LIN {X 0,Y 224.89,Z 892.917,A -85,B 0,C 180,E1 -24408.732,E2 -24408.732} C_VEL
LIN {X 0,Y 229.595,Z 886.207,A -85,B 0,C 180,E1 -24414.165,E2 -24414.165} C_VEL
LIN {X 0,Y 235.615,Z 877.788,A -85,B 0,C 180,E1 -24419.211,E2 -24419.211} C_VEL
LIN {X 0,Y 242.277,Z 868.356,A -85,B 0,C 180,E1 -24423.575,E2 -24423.575} C_VEL
LIN {X 0,Y 250.04,Z 856.97,A -85,B 0,C 180,E1 -24427.722,E2 -24427.722} C_VEL
LIN {X 0,Y 258.343,Z 844.109,A -85,B 0,C 180,E1 -24431.44,E2 -24431.44} C_VEL
LIN {X 0,Y 266.959,Z 829.748,A -85,B 0,C 180,E1 -24434.761,E2 -24434.761} C_VEL
LIN {X 0,Y 275.684,Z 813.801,A -85,B 0,C 180,E1 -24437.722,E2 -24437.722} C_VEL
LIN {X 0,Y 283.965,Z 796.943,A -85,B 0,C 180,E1 -24440.246,E2 -24440.246} C_VEL
LIN {X 0,Y 291.586,Z 779.329,A -85,B 0,C 180,E1 -24442.385,E2 -24442.385} C_VEL
LIN {X 0,Y 298.391,Z 761.127,A -85,B 0,C 180,E1 -24444.186,E2 -24444.186} C_VEL
LIN {X 0,Y 304.38,Z 742.174,A -85,B 0,C 180,E1 -24445.708,E2 -24445.708} C_VEL
LIN {X 0,Y 309.449,Z 722.453,A -85,B 0,C 180,E1 -24446.981,E2 -24446.981} C_VEL
LIN {X 0,Y 313.937,Z 699.919,A -85,B 0,C 180,E1 -24448.124,E2 -24448.124} C_VEL
LIN {X 0,Y 321.08,Z 660.976,A -85,B 0,C 180,E1 -24449.711,E2 -24449.711} C_VEL
LIN {X 0,Y 328.367,Z 619.459,A -85,B 0,C 180,E1 -24450.997,E2 -24450.997} C_VEL
LIN {X 0,Y 335.529,Z 572.373,A -85,B 0,C 180,E1 -24452.169,E2 -24452.169} C_VEL
LIN {X 0,Y 341.071,Z 525.516,A -85,B 0,C 180,E1 -24453.138,E2 -24453.138} C_VEL
LIN {X 0,Y 346.043,Z 470.407,A -85,B 0,C 180,E1 -24454.114,E2 -24454.114} C_VEL
LIN {X 0,Y 346.243,Z 465.398,A -85,B 0,C 180,E1 -24454.36,E2 -24454.36} C_VEL
LIN {X 0,Y 346.398,Z 453.089,A -85,B 0,C 180,E1 -24455.622,E2 -24455.622} C_VEL
LIN {X 0,Y 347.142,Z 448.885,A -85,B 0,C 180,E1 -24455.86,E2 -24455.86} C_VEL
LIN {X 0,Y 347.825,Z 446.041,A -85,B 0,C 180,E1 -24455.948,E2 -24455.948} C_VEL
LIN {X 0,Y 344.964,Z 434.776,A -85,B 0,C 180,E1 -24458.891,E2 -24458.891} C_VEL
LIN {X 0,Y 342.252,Z 424.826,A -85,B 0,C 180,E1 -24462.048,E2 -24462.048} C_VEL
LIN {X 0,Y 339.928,Z 416.846,A -85,B 0,C 180,E1 -24465.172,E2 -24465.172} C_VEL
LIN {X 0,Y 338.009,Z 410.266,A -85,B 0,C 180,E1 -24468.395,E2 -24468.395} C_VEL
LIN {X 0,Y 336.969,Z 406.588,A -85,B 0,C 180,E1 -24470.693,E2 -24470.693} C_VEL
LIN {X 0,Y 336.176,Z 403.515,A -85,B 0,C 180,E1 -24472.995,E2 -24472.995} C_VEL
LIN {X 0,Y 335.703,Z 399.838,A -85,B 0,C 180,E1 -24476.756,E2 -24476.756} C_VEL
LIN {X 0,Y 336.154,Z 398.855,A -85,B 0,C 180,E1 -24482.046,E2 -24482.046} C_VEL
LIN {X 0,Y 337.525,Z 399.846,A -85,B 0,C 180,E1 -24485.44,E2 -24485.44} C_VEL
LIN {X 0,Y 338.217,Z 411.43,A -85,B 0,C 180,E1 -24489.358,E2 -24489.358} C_VEL
LIN {X 0,Y 339.496,Z 420.899,A -85,B 0,C 180,E1 -24492.157,E2 -24492.157} C_VEL
LIN {X 0,Y 342.954,Z 437.759,A -85,B 0,C 180,E1 -24496.558,E2 -24496.558} C_VEL
LIN {X 0,Y 343.815,Z 442.334,A -85,B 0,C 180,E1 -24497.518,E2 -24497.518} C_VEL
LIN {X 0,Y 324.701,Z 558.02,A -85,B 0,C 180,E1 -24500.535,E2 -24500.535} C_VEL
LIN {X 0,Y 319.052,Z 621.611,A -85,B 0,C 180,E1 -24501.884,E2 -24501.884} C_VEL
LIN {X 0,Y 314.329,Z 657.117,A -85,B 0,C 180,E1 -24502.75,E2 -24502.75} C_VEL
LIN {X 0,Y 308.487,Z 691.069,A -85,B 0,C 180,E1 -24503.801,E2 -24503.801} C_VEL
LIN {X 0,Y 301.049,Z 726.478,A -85,B 0,C 180,E1 -24505.162,E2 -24505.162} C_VEL
LIN {X 0,Y 293.63,Z 757.559,A -85,B 0,C 180,E1 -24506.711,E2 -24506.711} C_VEL
LIN {X 0,Y 285.371,Z 788.213,A -85,B 0,C 180,E1 -24508.633,E2 -24508.633} C_VEL
LIN {X 0,Y 279.619,Z 806.503,A -85,B 0,C 180,E1 -24510.076,E2 -24510.076} C_VEL
LIN {X 0,Y 272.693,Z 824.978,A -85,B 0,C 180,E1 -24511.871,E2 -24511.871} C_VEL
LIN {X 0,Y 264.997,Z 842.919,A -85,B 0,C 180,E1 -24514.053,E2 -24514.053} C_VEL
LIN {X 0,Y 256.789,Z 860.091,A -85,B 0,C 180,E1 -24516.666,E2 -24516.666} C_VEL
LIN {X 0,Y 248.598,Z 875.732,A -85,B 0,C 180,E1 -24519.625,E2 -24519.625} C_VEL
LIN {X 0,Y 240.08,Z 890.924,A -85,B 0,C 180,E1 -24523.211,E2 -24523.211} C_VEL
LIN {X 0,Y 232.336,Z 904.2,A -85,B 0,C 180,E1 -24527.159,E2 -24527.159} C_VEL
LIN {X 0,Y 225.293,Z 916.132,A -85,B 0,C 180,E1 -24531.586,E2 -24531.586} C_VEL
LIN {X 0,Y 219.007,Z 927.216,A -85,B 0,C 180,E1 -24536.779,E2 -24536.779} C_VEL
LIN {X 0,Y 214.367,Z 936.293,A -85,B 0,C 180,E1 -24542.197,E2 -24542.197} C_VEL
LIN {X 0,Y 211.27,Z 943.925,A -85,B 0,C 180,E1 -24548.068,E2 -24548.068} C_VEL
LIN {X 0,Y 209.887,Z 949.622,A -85,B 0,C 180,E1 -24553.96,E2 -24553.96} C_VEL
LIN {X 0,Y 209.829,Z 953.456,A -85,B 0,C 180,E1 -24559.567,E2 -24559.567} C_VEL
LIN {X 0,Y 210.451,Z 955.606,A -85,B 0,C 180,E1 -24564.547,E2 -24564.547} C_VEL
LIN {X 0,Y 210.953,Z 956.378,A -85,B 0,C 180,E1 -24568.914,E2 -24568.914} C_VEL
LIN {X 0,Y 210.827,Z 956.176,A -85,B 0,C 180,E1 -24572.991,E2 -24572.991} C_VEL
LIN {X 0,Y 210.324,Z 955.42,A -85,B 0,C 180,E1 -24576.826,E2 -24576.826} C_VEL
LIN {X 0,Y 209.602,Z 955.36,A -85,B 0,C 180,E1 -24582.396,E2 -24582.396} C_VEL
LIN {X 0,Y 210.22,Z 953.841,A -85,B 0,C 180,E1 -24589.159,E2 -24589.159} C_VEL
LIN {X 0,Y 214.082,Z 950.092,A -85,B 0,C 180,E1 -24597.24,E2 -24597.24} C_VEL
LIN {X 0,Y 222.093,Z 944.496,A -85,B 0,C 180,E1 -24605.189,E2 -24605.189} C_VEL
LIN {X 0,Y 235.722,Z 936.412,A -85,B 0,C 180,E1 -24613.147,E2 -24613.147} C_VEL
LIN {X 0,Y 254.87,Z 926.374,A -85,B 0,C 180,E1 -24620.259,E2 -24620.259} C_VEL
LIN {X 0,Y 266.015,Z 920.808,A -85,B 0,C 180,E1 -24623.298,E2 -24623.298} C_VEL
LIN {X 0,Y 250.517,Z 923.428,A -85,B 0,C 180,E1 -24627.796,E2 -24627.796} C_VEL
LIN {X 0,Y 237.812,Z 924.193,A -85,B 0,C 180,E1 -24632.723,E2 -24632.723} C_VEL
LIN {X 0,Y 228.43,Z 923.252,A -85,B 0,C 180,E1 -24637.615,E2 -24637.615} C_VEL
LIN {X 0,Y 221.072,Z 920.618,A -85,B 0,C 180,E1 -24642.903,E2 -24642.903} C_VEL
LIN {X 0,Y 215.973,Z 916.354,A -85,B 0,C 180,E1 -24648.246,E2 -24648.246} C_VEL
LIN {X 0,Y 212.767,Z 910.583,A -85,B 0,C 180,E1 -24653.524,E2 -24653.524} C_VEL
LIN {X 0,Y 211.014,Z 902.853,A -85,B 0,C 180,E1 -24658.944,E2 -24658.944} C_VEL
LIN {X 0,Y 210.442,Z 893.66,A -85,B 0,C 180,E1 -24664.087,E2 -24664.087} C_VEL
LIN {X 0,Y 210.785,Z 882.923,A -85,B 0,C 180,E1 -24669.006,E2 -24669.006} C_VEL
LIN {X 0,Y 211.915,Z 870.762,A -85,B 0,C 180,E1 -24673.646,E2 -24673.646} C_VEL
LIN {X 0,Y 213.952,Z 856.352,A -85,B 0,C 180,E1 -24678.247,E2 -24678.247} C_VEL
LIN {X 0,Y 216.755,Z 840.361,A -85,B 0,C 180,E1 -24682.512,E2 -24682.512} C_VEL
LIN {X 0,Y 218.378,Z 832.199,A -85,B 0,C 180,E1 -24684.48,E2 -24684.48} C_VEL
LIN {X 0,Y 220.054,Z 831.839,A -85,B 0,C 180,E1 -24685.573,E2 -24685.573} C_VEL
LIN {X 0,Y 223.639,Z 829.907,A -85,B 0,C 180,E1 -24686.845,E2 -24686.845} C_VEL
LIN {X 0,Y 226.592,Z 828.838,A -85,B 0,C 180,E1 -24688.175,E2 -24688.175} C_VEL
LIN {X 0,Y 230.34,Z 826.932,A -85,B 0,C 180,E1 -24689.375,E2 -24689.375} C_VEL
LIN {X 0,Y 234.504,Z 825.124,A -85,B 0,C 180,E1 -24690.775,E2 -24690.775} C_VEL
LIN {X 0,Y 237.283,Z 823.677,A -85,B 0,C 180,E1 -24691.502,E2 -24691.502} C_VEL
LIN {X 0,Y 242.468,Z 821.37,A -85,B 0,C 180,E1 -24692.98,E2 -24692.98} C_VEL
LIN {X 0,Y 246.111,Z 819.479,A -85,B 0,C 180,E1 -24693.821,E2 -24693.821} C_VEL
LIN {X 0,Y 252.074,Z 816.571,A -85,B 0,C 180,E1 -24695.201,E2 -24695.201} C_VEL
LIN {X 0,Y 255.675,Z 814.634,A -85,B 0,C 180,E1 -24695.918,E2 -24695.918} C_VEL
LIN {X 0,Y 262.61,Z 811.083,A -85,B 0,C 180,E1 -24697.258,E2 -24697.258} C_VEL
LIN {X 0,Y 267.555,Z 808.331,A -85,B 0,C 180,E1 -24698.071,E2 -24698.071} C_VEL
LIN {X 0,Y 275.109,Z 804.086,A -85,B 0,C 180,E1 -24699.228,E2 -24699.228} C_VEL
LIN {X 0,Y 276.135,Z 803.504,A -85,B 0,C 180,E1 -24699.382,E2 -24699.382} C_VEL
LIN {X 0,Y 267.372,Z 820.191,A -85,B 0,C 180,E1 -24702.069,E2 -24702.069} C_VEL
LIN {X 0,Y 258.262,Z 835.758,A -85,B 0,C 180,E1 -24705.2,E2 -24705.2} C_VEL
LIN {X 0,Y 249.569,Z 849.375,A -85,B 0,C 180,E1 -24708.618,E2 -24708.618} C_VEL
LIN {X 0,Y 240.778,Z 862.18,A -85,B 0,C 180,E1 -24712.677,E2 -24712.677} C_VEL
LIN {X 0,Y 233.059,Z 872.853,A -85,B 0,C 180,E1 -24716.984,E2 -24716.984} C_VEL
LIN {X 0,Y 226.167,Z 882.078,A -85,B 0,C 180,E1 -24721.767,E2 -24721.767} C_VEL
LIN {X 0,Y 220.376,Z 889.781,A -85,B 0,C 180,E1 -24727.033,E2 -24727.033} C_VEL
LIN {X 0,Y 216.078,Z 895.64,A -85,B 0,C 180,E1 -24732.495,E2 -24732.495} C_VEL
LIN {X 0,Y 213.212,Z 899.787,A -85,B 0,C 180,E1 -24738.092,E2 -24738.092} C_VEL
LIN {X 0,Y 211.636,Z 902.278,A -85,B 0,C 180,E1 -24743.761,E2 -24743.761} C_VEL
LIN {X 0,Y 211.092,Z 903.177,A -85,B 0,C 180,E1 -24749.186,E2 -24749.186} C_VEL
LIN {X 0,Y 211.364,Z 902.697,A -85,B 0,C 180,E1 -24754.613,E2 -24754.613} C_VEL
LIN {X 0,Y 212.614,Z 900.69,A -85,B 0,C 180,E1 -24760.294,E2 -24760.294} C_VEL
LIN {X 0,Y 215.071,Z 897.086,A -85,B 0,C 180,E1 -24765.92,E2 -24765.92} C_VEL
LIN {X 0,Y 218.936,Z 891.789,A -85,B 0,C 180,E1 -24771.43,E2 -24771.43} C_VEL
LIN {X 0,Y 224,Z 885.074,A -85,B 0,C 180,E1 -24776.512,E2 -24776.512} C_VEL
LIN {X 0,Y 230.407,Z 876.576,A -85,B 0,C 180,E1 -24781.383,E2 -24781.383} C_VEL
LIN {X 0,Y 238.113,Z 866.087,A -85,B 0,C 180,E1 -24786.007,E2 -24786.007} C_VEL
LIN {X 0,Y 246.102,Z 854.75,A -85,B 0,C 180,E1 -24789.937,E2 -24789.937} C_VEL
LIN {X 0,Y 254.985,Z 841.256,A -85,B 0,C 180,E1 -24793.643,E2 -24793.643} C_VEL
LIN {X 0,Y 263.722,Z 826.902,A -85,B 0,C 180,E1 -24796.796,E2 -24796.796} C_VEL
LIN {X 0,Y 272.5,Z 810.986,A -85,B 0,C 180,E1 -24799.609,E2 -24799.609} C_VEL
LIN {X 0,Y 280.898,Z 793.934,A -85,B 0,C 180,E1 -24802.041,E2 -24802.041} C_VEL
LIN {X 0,Y 288.397,Z 776.609,A -85,B 0,C 180,E1 -24804.053,E2 -24804.053} C_VEL
LIN {X 0,Y 295.434,Z 757.617,A -85,B 0,C 180,E1 -24805.843,E2 -24805.843} C_VEL
LIN {X 0,Y 301.413,Z 738.331,A -85,B 0,C 180,E1 -24807.305,E2 -24807.305} C_VEL
LIN {X 0,Y 306.434,Z 718.043,A -85,B 0,C 180,E1 -24808.534,E2 -24808.534} C_VEL
LIN {X 0,Y 313.749,Z 680.473,A -85,B 0,C 180,E1 -24810.254,E2 -24810.254} C_VEL
LIN {X 0,Y 321.162,Z 640.371,A -85,B 0,C 180,E1 -24811.667,E2 -24811.667} C_VEL
LIN {X 0,Y 328.989,Z 593.753,A -85,B 0,C 180,E1 -24812.913,E2 -24812.913} C_VEL
LIN {X 0,Y 335.28,Z 547.106,A -85,B 0,C 180,E1 -24813.943,E2 -24813.943} C_VEL
LIN {X 0,Y 340.536,Z 494.772,A -85,B 0,C 180,E1 -24814.91,E2 -24814.91} C_VEL
LIN {X 0,Y 343.544,Z 463.899,A -85,B 0,C 180,E1 -24815.454,E2 -24815.454} C_VEL
LIN {X 0,Y 347.142,Z 448.885,A -85,B 0,C 180,E1 -24815.86,E2 -24815.86} C_VEL
LIN {X 0,Y 347.548,Z 445.802,A -85,B 0,C 180,E1 -24816.106,E2 -24816.106} C_VEL
LIN {X 0,Y 347.187,Z 442.834,A -85,B 0,C 180,E1 -24816.678,E2 -24816.678} C_VEL
LIN {X 0,Y 345.794,Z 440.355,A -85,B 0,C 180,E1 -24817.666,E2 -24817.666} C_VEL
LIN {X 0,Y 341.285,Z 437.262,A -85,B 0,C 180,E1 -24820.497,E2 -24820.497} C_VEL
LIN {X 0,Y 340.469,Z 435.442,A -85,B 0,C 180,E1 -24821.294,E2 -24821.294} C_VEL
LIN {X 0,Y 338.282,Z 427.186,A -85,B 0,C 180,E1 -24824.265,E2 -24824.265} C_VEL
LIN {X 0,Y 336.371,Z 420.098,A -85,B 0,C 180,E1 -24827.467,E2 -24827.467} C_VEL
LIN {X 0,Y 335.021,Z 414.87,A -85,B 0,C 180,E1 -24830.379,E2 -24830.379} C_VEL
LIN {X 0,Y 334.091,Z 411.077,A -85,B 0,C 180,E1 -24833.297,E2 -24833.297} C_VEL
LIN {X 0,Y 333.789,Z 407.578,A -85,B 0,C 180,E1 -24836.909,E2 -24836.909} C_VEL
LIN {X 0,Y 334.325,Z 406.643,A -85,B 0,C 180,E1 -24842.057,E2 -24842.057} C_VEL
LIN {X 0,Y 335.554,Z 407.569,A -85,B 0,C 180,E1 -24845.129,E2 -24845.129} C_VEL
LIN {X 0,Y 336.427,Z 420.93,A -85,B 0,C 180,E1 -24849.624,E2 -24849.624} C_VEL
LIN {X 0,Y 339.49,Z 440.436,A -85,B 0,C 180,E1 -24854.973,E2 -24854.973} C_VEL
LIN {X 0,Y 340.649,Z 446.205,A -85,B 0,C 180,E1 -24856.334,E2 -24856.334} C_VEL
LIN {X 0,Y 322.123,Z 555.167,A -85,B 0,C 180,E1 -24859.143,E2 -24859.143} C_VEL
LIN {X 0,Y 316.244,Z 619.304,A -85,B 0,C 180,E1 -24860.5,E2 -24860.5} C_VEL
LIN {X 0,Y 311.347,Z 655.198,A -85,B 0,C 180,E1 -24861.357,E2 -24861.357} C_VEL
LIN {X 0,Y 305.407,Z 688.827,A -85,B 0,C 180,E1 -24862.379,E2 -24862.379} C_VEL
LIN {X 0,Y 297.92,Z 723.828,A -85,B 0,C 180,E1 -24863.691,E2 -24863.691} C_VEL
LIN {X 0,Y 290.514,Z 754.277,A -85,B 0,C 180,E1 -24865.151,E2 -24865.151} C_VEL
LIN {X 0,Y 281.87,Z 785.806,A -85,B 0,C 180,E1 -24867.079,E2 -24867.079} C_VEL
LIN {X 0,Y 275.545,Z 805.229,A -85,B 0,C 180,E1 -24868.579,E2 -24868.579} C_VEL
LIN {X 0,Y 267.973,Z 824.701,A -85,B 0,C 180,E1 -24870.466,E2 -24870.466} C_VEL
LIN {X 0,Y 260.035,Z 842.471,A -85,B 0,C 180,E1 -24872.637,E2 -24872.637} C_VEL
LIN {X 0,Y 251.6,Z 859.39,A -85,B 0,C 180,E1 -24875.226,E2 -24875.226} C_VEL
LIN {X 0,Y 242.748,Z 875.525,A -85,B 0,C 180,E1 -24878.309,E2 -24878.309} C_VEL
LIN {X 0,Y 233.873,Z 890.528,A -85,B 0,C 180,E1 -24881.935,E2 -24881.935} C_VEL
LIN {X 0,Y 225.322,Z 904.412,A -85,B 0,C 180,E1 -24886.19,E2 -24886.19} C_VEL
LIN {X 0,Y 217.625,Z 916.766,A -85,B 0,C 180,E1 -24890.99,E2 -24890.99} C_VEL
LIN {X 0,Y 211.432,Z 927.087,A -85,B 0,C 180,E1 -24896.08,E2 -24896.08} C_VEL
LIN {X 0,Y 206.508,Z 936.172,A -85,B 0,C 180,E1 -24901.791,E2 -24901.791} C_VEL
LIN {X 0,Y 203.356,Z 943.418,A -85,B 0,C 180,E1 -24907.753,E2 -24907.753} C_VEL
LIN {X 0,Y 201.913,Z 948.996,A -85,B 0,C 180,E1 -24913.9,E2 -24913.9} C_VEL
LIN {X 0,Y 201.905,Z 952.845,A -85,B 0,C 180,E1 -24920.019,E2 -24920.019} C_VEL
LIN {X 0,Y 202.637,Z 954.84,A -85,B 0,C 180,E1 -24925.38,E2 -24925.38} C_VEL
LIN {X 0,Y 203.037,Z 955.434,A -85,B 0,C 180,E1 -24929.718,E2 -24929.718} C_VEL
LIN {X 0,Y 202.771,Z 954.989,A -85,B 0,C 180,E1 -24933.959,E2 -24933.959} C_VEL
LIN {X 0,Y 202.19,Z 953.885,A -85,B 0,C 180,E1 -24938.532,E2 -24938.532} C_VEL
LIN {X 0,Y 201.691,Z 953.677,A -85,B 0,C 180,E1 -24944.352,E2 -24944.352} C_VEL
LIN {X 0,Y 202.951,Z 952.051,A -85,B 0,C 180,E1 -24951.384,E2 -24951.384} C_VEL
LIN {X 0,Y 208.335,Z 947.988,A -85,B 0,C 180,E1 -24960.261,E2 -24960.261} C_VEL
LIN {X 0,Y 218.347,Z 942.174,A -85,B 0,C 180,E1 -24968.521,E2 -24968.521} C_VEL
LIN {X 0,Y 234.358,Z 934.019,A -85,B 0,C 180,E1 -24976.495,E2 -24976.495} C_VEL
LIN {X 0,Y 254.283,Z 924.78,A -85,B 0,C 180,E1 -24982.962,E2 -24982.962} C_VEL
LIN {X 0,Y 255.683,Z 924.14,A -85,B 0,C 180,E1 -24983.389,E2 -24983.389} C_VEL
LIN {X 0,Y 240.072,Z 925.76,A -85,B 0,C 180,E1 -24988.174,E2 -24988.174} C_VEL
LIN {X 0,Y 228.015,Z 925.552,A -85,B 0,C 180,E1 -24993.149,E2 -24993.149} C_VEL
LIN {X 0,Y 218.832,Z 923.767,A -85,B 0,C 180,E1 -24998.278,E2 -24998.278} C_VEL
LIN {X 0,Y 212.032,Z 920.47,A -85,B 0,C 180,E1 -25003.564,E2 -25003.564} C_VEL
LIN {X 0,Y 207.169,Z 915.443,A -85,B 0,C 180,E1 -25009.15,E2 -25009.15} C_VEL
LIN {X 0,Y 204.129,Z 908.473,A -85,B 0,C 180,E1 -25014.942,E2 -25014.942} C_VEL
LIN {X 0,Y 202.762,Z 900.32,A -85,B 0,C 180,E1 -25020.283,E2 -25020.283} C_VEL
LIN {X 0,Y 202.452,Z 890.814,A -85,B 0,C 180,E1 -25025.385,E2 -25025.385} C_VEL
LIN {X 0,Y 203.044,Z 879.3,A -85,B 0,C 180,E1 -25030.498,E2 -25030.498} C_VEL
LIN {X 0,Y 204.494,Z 866.311,A -85,B 0,C 180,E1 -25035.31,E2 -25035.31} C_VEL
LIN {X 0,Y 206.922,Z 850.934,A -85,B 0,C 180,E1 -25040.065,E2 -25040.065} C_VEL
LIN {X 0,Y 208.98,Z 840.037,A -85,B 0,C 180,E1 -25043.026,E2 -25043.026} C_VEL
LIN {X 0,Y 210.871,Z 839.52,A -85,B 0,C 180,E1 -25044.364,E2 -25044.364} C_VEL
LIN {X 0,Y 213.774,Z 837.959,A -85,B 0,C 180,E1 -25045.488,E2 -25045.488} C_VEL
LIN {X 0,Y 216.495,Z 837.046,A -85,B 0,C 180,E1 -25046.912,E2 -25046.912} C_VEL
LIN {X 0,Y 220.034,Z 835.344,A -85,B 0,C 180,E1 -25048.204,E2 -25048.204} C_VEL
LIN {X 0,Y 223.983,Z 833.719,A -85,B 0,C 180,E1 -25049.704,E2 -25049.704} C_VEL
LIN {X 0,Y 226.594,Z 832.46,A -85,B 0,C 180,E1 -25050.495,E2 -25050.495} C_VEL
LIN {X 0,Y 231.577,Z 830.349,A -85,B 0,C 180,E1 -25052.079,E2 -25052.079} C_VEL
LIN {X 0,Y 234.959,Z 828.778,A -85,B 0,C 180,E1 -25053.005,E2 -25053.005} C_VEL
LIN {X 0,Y 241.29,Z 825.829,A -85,B 0,C 180,E1 -25054.592,E2 -25054.592} C_VEL
LIN {X 0,Y 250.192,Z 821.605,A -85,B 0,C 180,E1 -25056.554,E2 -25056.554} C_VEL
LIN {X 0,Y 261.296,Z 816.099,A -85,B 0,C 180,E1 -25058.59,E2 -25058.59} C_VEL
LIN {X 0,Y 266.545,Z 813.328,A -85,B 0,C 180,E1 -25059.413,E2 -25059.413} C_VEL
LIN {X 0,Y 257.171,Z 829.628,A -85,B 0,C 180,E1 -25062.377,E2 -25062.377} C_VEL
LIN {X 0,Y 247.802,Z 844.317,A -85,B 0,C 180,E1 -25065.728,E2 -25065.728} C_VEL
LIN {X 0,Y 238.695,Z 857.461,A -85,B 0,C 180,E1 -25069.512,E2 -25069.512} C_VEL
LIN {X 0,Y 230.087,Z 869.099,A -85,B 0,C 180,E1 -25073.771,E2 -25073.771} C_VEL
LIN {X 0,Y 222.258,Z 879.206,A -85,B 0,C 180,E1 -25078.543,E2 -25078.543} C_VEL
LIN {X 0,Y 215.768,Z 887.387,A -85,B 0,C 180,E1 -25083.585,E2 -25083.585} C_VEL
LIN {X 0,Y 210.469,Z 894.092,A -85,B 0,C 180,E1 -25089.126,E2 -25089.126} C_VEL
LIN {X 0,Y 206.702,Z 899.028,A -85,B 0,C 180,E1 -25094.857,E2 -25094.857} C_VEL
LIN {X 0,Y 204.391,Z 902.303,A -85,B 0,C 180,E1 -25100.709,E2 -25100.709} C_VEL
LIN {X 0,Y 203.309,Z 903.961,A -85,B 0,C 180,E1 -25106.616,E2 -25106.616} C_VEL
LIN {X 0,Y 203.212,Z 904.09,A -85,B 0,C 180,E1 -25112.256,E2 -25112.256} C_VEL
LIN {X 0,Y 204.008,Z 902.842,A -85,B 0,C 180,E1 -25117.888,E2 -25117.888} C_VEL
LIN {X 0,Y 206.112,Z 899.833,A -85,B 0,C 180,E1 -25124.037,E2 -25124.037} C_VEL
LIN {X 0,Y 209.786,Z 895.013,A -85,B 0,C 180,E1 -25130.07,E2 -25130.07} C_VEL
LIN {X 0,Y 214.836,Z 888.617,A -85,B 0,C 180,E1 -25135.648,E2 -25135.648} C_VEL
LIN {X 0,Y 221.454,Z 880.322,A -85,B 0,C 180,E1 -25140.979,E2 -25140.979} C_VEL
LIN {X 0,Y 229.143,Z 870.475,A -85,B 0,C 180,E1 -25145.783,E2 -25145.783} C_VEL
LIN {X 0,Y 237.624,Z 859.12,A -85,B 0,C 180,E1 -25150.076,E2 -25150.076} C_VEL
LIN {X 0,Y 246.624,Z 846.271,A -85,B 0,C 180,E1 -25153.891,E2 -25153.891} C_VEL
LIN {X 0,Y 255.338,Z 832.826,A -85,B 0,C 180,E1 -25157.078,E2 -25157.078} C_VEL
LIN {X 0,Y 264.272,Z 817.707,A -85,B 0,C 180,E1 -25159.968,E2 -25159.968} C_VEL
LIN {X 0,Y 272.923,Z 801.409,A -85,B 0,C 180,E1 -25162.483,E2 -25162.483} C_VEL
LIN {X 0,Y 281.204,Z 783.726,A -85,B 0,C 180,E1 -25164.691,E2 -25164.691} C_VEL
LIN {X 0,Y 288.732,Z 765.064,A -85,B 0,C 180,E1 -25166.573,E2 -25166.573} C_VEL
LIN {X 0,Y 295.016,Z 746.597,A -85,B 0,C 180,E1 -25168.08,E2 -25168.08} C_VEL
LIN {X 0,Y 300.676,Z 726.186,A -85,B 0,C 180,E1 -25169.416,E2 -25169.416} C_VEL
LIN {X 0,Y 305.859,Z 701.959,A -85,B 0,C 180,E1 -25170.65,E2 -25170.65} C_VEL
LIN {X 0,Y 313.548,Z 662.516,A -85,B 0,C 180,E1 -25172.245,E2 -25172.245} C_VEL
LIN {X 0,Y 320.97,Z 622.102,A -85,B 0,C 180,E1 -25173.476,E2 -25173.476} C_VEL
LIN {X 0,Y 328.272,Z 576.098,A -85,B 0,C 180,E1 -25174.596,E2 -25174.596} C_VEL
LIN {X 0,Y 333.972,Z 529.706,A -85,B 0,C 180,E1 -25175.533,E2 -25175.533} C_VEL
LIN {X 0,Y 340.15,Z 466.539,A -85,B 0,C 180,E1 -25176.644,E2 -25176.644} C_VEL
LIN {X 0,Y 344.086,Z 450.132,A -85,B 0,C 180,E1 -25177.099,E2 -25177.099} C_VEL
LIN {X 0,Y 341.351,Z 438.925,A -85,B 0,C 180,E1 -25180.18,E2 -25180.18} C_VEL
LIN {X 0,Y 340.469,Z 435.442,A -85,B 0,C 180,E1 -25181.294,E2 -25181.294} C_VEL
LIN {X 0,Y 339.282,Z 432.899,A -85,B 0,C 180,E1 -25182.512,E2 -25182.512} C_VEL
LIN {X 0,Y 336.733,Z 431.213,A -85,B 0,C 180,E1 -25184.633,E2 -25184.633} C_VEL
LIN {X 0,Y 334.628,Z 429.482,A -85,B 0,C 180,E1 -25186.699,E2 -25186.699} C_VEL
LIN {X 0,Y 334.307,Z 428.715,A -85,B 0,C 180,E1 -25187.159,E2 -25187.159} C_VEL
LIN {X 0,Y 332.924,Z 422.507,A -85,B 0,C 180,E1 -25190.579,E2 -25190.579} C_VEL
LIN {X 0,Y 332.056,Z 418.778,A -85,B 0,C 180,E1 -25193.429,E2 -25193.429} C_VEL
LIN {X 0,Y 331.825,Z 415.306,A -85,B 0,C 180,E1 -25197.064,E2 -25197.064} C_VEL
LIN {X 0,Y 332.528,Z 414.439,A -85,B 0,C 180,E1 -25202.068,E2 -25202.068} C_VEL
LIN {X 0,Y 333.593,Z 415.275,A -85,B 0,C 180,E1 -25204.814,E2 -25204.814} C_VEL
LIN {X 0,Y 334.377,Z 429.017,A -85,B 0,C 180,E1 -25209.379,E2 -25209.379} C_VEL
LIN {X 0,Y 337.146,Z 447.925,A -85,B 0,C 180,E1 -25214.557,E2 -25214.557} C_VEL
LIN {X 0,Y 337.566,Z 450.515,A -85,B 0,C 180,E1 -25215.139,E2 -25215.139} C_VEL
LIN {X 0,Y 319.756,Z 552.113,A -85,B 0,C 180,E1 -25217.726,E2 -25217.726} C_VEL
LIN {X 0,Y 313.651,Z 616.805,A -85,B 0,C 180,E1 -25219.088,E2 -25219.088} C_VEL
LIN {X 0,Y 308.573,Z 653.152,A -85,B 0,C 180,E1 -25219.934,E2 -25219.934} C_VEL
LIN {X 0,Y 302.296,Z 687.872,A -85,B 0,C 180,E1 -25220.968,E2 -25220.968} C_VEL
LIN {X 0,Y 294.883,Z 721.646,A -85,B 0,C 180,E1 -25222.211,E2 -25222.211} C_VEL
LIN {X 0,Y 287.35,Z 751.98,A -85,B 0,C 180,E1 -25223.616,E2 -25223.616} C_VEL
LIN {X 0,Y 278.355,Z 784.046,A -85,B 0,C 180,E1 -25225.535,E2 -25225.535} C_VEL
LIN {X 0,Y 272.028,Z 802.983,A -85,B 0,C 180,E1 -25226.956,E2 -25226.956} C_VEL
LIN {X 0,Y 264.192,Z 822.641,A -85,B 0,C 180,E1 -25228.818,E2 -25228.818} C_VEL
LIN {X 0,Y 255.628,Z 841.24,A -85,B 0,C 180,E1 -25231.061,E2 -25231.061} C_VEL
LIN {X 0,Y 246.829,Z 858.228,A -85,B 0,C 180,E1 -25233.647,E2 -25233.647} C_VEL
LIN {X 0,Y 237.72,Z 874.11,A -85,B 0,C 180,E1 -25236.675,E2 -25236.675} C_VEL
LIN {X 0,Y 228.326,Z 889.305,A -85,B 0,C 180,E1 -25240.361,E2 -25240.361} C_VEL
LIN {X 0,Y 219.526,Z 902.891,A -85,B 0,C 180,E1 -25244.543,E2 -25244.543} C_VEL
LIN {X 0,Y 211.133,Z 915.618,A -85,B 0,C 180,E1 -25249.548,E2 -25249.548} C_VEL
LIN {X 0,Y 204.191,Z 926.472,A -85,B 0,C 180,E1 -25255.045,E2 -25255.045} C_VEL
LIN {X 0,Y 198.818,Z 935.674,A -85,B 0,C 180,E1 -25261.132,E2 -25261.132} C_VEL
LIN {X 0,Y 195.438,Z 942.931,A -85,B 0,C 180,E1 -25267.436,E2 -25267.436} C_VEL
LIN {X 0,Y 193.909,Z 948.606,A -85,B 0,C 180,E1 -25274.14,E2 -25274.14} C_VEL
LIN {X 0,Y 193.96,Z 952.104,A -85,B 0,C 180,E1 -25280.205,E2 -25280.205} C_VEL
LIN {X 0,Y 194.718,Z 953.916,A -85,B 0,C 180,E1 -25285.583,E2 -25285.583} C_VEL
LIN {X 0,Y 195.109,Z 954.446,A -85,B 0,C 180,E1 -25290,E2 -25290} C_VEL
LIN {X 0,Y 194.783,Z 953.918,A -85,B 0,C 180,E1 -25294.416,E2 -25294.416} C_VEL
LIN {X 0,Y 194.115,Z 952.266,A -85,B 0,C 180,E1 -25300.087,E2 -25300.087} C_VEL
LIN {X 0,Y 193.988,Z 951.89,A -85,B 0,C 180,E1 -25306.777,E2 -25306.777} C_VEL
LIN {X 0,Y 196.359,Z 949.933,A -85,B 0,C 180,E1 -25314.681,E2 -25314.681} C_VEL
LIN {X 0,Y 203.821,Z 945.545,A -85,B 0,C 180,E1 -25324.004,E2 -25324.004} C_VEL
LIN {X 0,Y 216.327,Z 939.485,A -85,B 0,C 180,E1 -25332.441,E2 -25332.441} C_VEL
LIN {X 0,Y 235.213,Z 931.168,A -85,B 0,C 180,E1 -25340.303,E2 -25340.303} C_VEL
LIN {X 0,Y 245.482,Z 926.927,A -85,B 0,C 180,E1 -25343.43,E2 -25343.43} C_VEL
LIN {X 0,Y 230.871,Z 927.562,A -85,B 0,C 180,E1 -25348.104,E2 -25348.104} C_VEL
LIN {X 0,Y 218.657,Z 926.56,A -85,B 0,C 180,E1 -25353.375,E2 -25353.375} C_VEL
LIN {X 0,Y 209.607,Z 924.018,A -85,B 0,C 180,E1 -25358.743,E2 -25358.743} C_VEL
LIN {X 0,Y 202.738,Z 919.727,A -85,B 0,C 180,E1 -25364.554,E2 -25364.554} C_VEL
LIN {X 0,Y 198.06,Z 913.469,A -85,B 0,C 180,E1 -25370.703,E2 -25370.703} C_VEL
LIN {X 0,Y 195.581,Z 905.888,A -85,B 0,C 180,E1 -25376.483,E2 -25376.483} C_VEL
LIN {X 0,Y 194.576,Z 897.367,A -85,B 0,C 180,E1 -25381.767,E2 -25381.767} C_VEL
LIN {X 0,Y 194.552,Z 887.031,A -85,B 0,C 180,E1 -25387.085,E2 -25387.085} C_VEL
LIN {X 0,Y 195.453,Z 874.895,A -85,B 0,C 180,E1 -25392.282,E2 -25392.282} C_VEL
LIN {X 0,Y 197.218,Z 861.476,A -85,B 0,C 180,E1 -25397.101,E2 -25397.101} C_VEL
LIN {X 0,Y 199.677,Z 847.469,A -85,B 0,C 180,E1 -25401.442,E2 -25401.442} C_VEL
LIN {X 0,Y 201.324,Z 847.012,A -85,B 0,C 180,E1 -25402.792,E2 -25402.792} C_VEL
LIN {X 0,Y 204.017,Z 845.607,A -85,B 0,C 180,E1 -25404.003,E2 -25404.003} C_VEL
LIN {X 0,Y 206.542,Z 844.763,A -85,B 0,C 180,E1 -25405.522,E2 -25405.522} C_VEL
LIN {X 0,Y 209.844,Z 843.247,A -85,B 0,C 180,E1 -25406.915,E2 -25406.915} C_VEL
LIN {X 0,Y 213.572,Z 841.761,A -85,B 0,C 180,E1 -25408.525,E2 -25408.525} C_VEL
LIN {X 0,Y 215.992,Z 840.669,A -85,B 0,C 180,E1 -25409.387,E2 -25409.387} C_VEL
LIN {X 0,Y 220.769,Z 838.719,A -85,B 0,C 180,E1 -25411.086,E2 -25411.086} C_VEL
LIN {X 0,Y 229.354,Z 835.015,A -85,B 0,C 180,E1 -25413.624,E2 -25413.624} C_VEL
LIN {X 0,Y 237.845,Z 831.343,A -85,B 0,C 180,E1 -25415.757,E2 -25415.757} C_VEL
LIN {X 0,Y 247.768,Z 826.829,A -85,B 0,C 180,E1 -25417.837,E2 -25417.837} C_VEL
LIN {X 0,Y 256.771,Z 822.752,A -85,B 0,C 180,E1 -25419.504,E2 -25419.504} C_VEL
LIN {X 0,Y 247.225,Z 837.953,A -85,B 0,C 180,E1 -25422.6,E2 -25422.6} C_VEL
LIN {X 0,Y 237.316,Z 852.257,A -85,B 0,C 180,E1 -25426.291,E2 -25426.291} C_VEL
LIN {X 0,Y 228.297,Z 864.319,A -85,B 0,C 180,E1 -25430.249,E2 -25430.249} C_VEL
LIN {X 0,Y 219.841,Z 874.97,A -85,B 0,C 180,E1 -25434.716,E2 -25434.716} C_VEL
LIN {X 0,Y 212.23,Z 884.171,A -85,B 0,C 180,E1 -25439.727,E2 -25439.727} C_VEL
LIN {X 0,Y 205.696,Z 891.933,A -85,B 0,C 180,E1 -25445.369,E2 -25445.369} C_VEL
LIN {X 0,Y 200.728,Z 897.907,A -85,B 0,C 180,E1 -25451.409,E2 -25451.409} C_VEL
LIN {X 0,Y 197.535,Z 901.951,A -85,B 0,C 180,E1 -25457.428,E2 -25457.428} C_VEL
LIN {X 0,Y 195.79,Z 904.377,A -85,B 0,C 180,E1 -25463.549,E2 -25463.549} C_VEL
LIN {X 0,Y 195.217,Z 905.198,A -85,B 0,C 180,E1 -25469.413,E2 -25469.413} C_VEL
LIN {X 0,Y 195.576,Z 904.642,A -85,B 0,C 180,E1 -25475.28,E2 -25475.28} C_VEL
LIN {X 0,Y 197.067,Z 902.567,A -85,B 0,C 180,E1 -25481.413,E2 -25481.413} C_VEL
LIN {X 0,Y 200.126,Z 898.677,A -85,B 0,C 180,E1 -25487.744,E2 -25487.744} C_VEL
LIN {X 0,Y 204.905,Z 892.926,A -85,B 0,C 180,E1 -25493.892,E2 -25493.892} C_VEL
LIN {X 0,Y 211.121,Z 885.568,A -85,B 0,C 180,E1 -25499.508,E2 -25499.508} C_VEL
LIN {X 0,Y 218.51,Z 876.704,A -85,B 0,C 180,E1 -25504.57,E2 -25504.57} C_VEL
LIN {X 0,Y 226.846,Z 866.319,A -85,B 0,C 180,E1 -25509.124,E2 -25509.124} C_VEL
LIN {X 0,Y 235.805,Z 854.497,A -85,B 0,C 180,E1 -25513.169,E2 -25513.169} C_VEL
LIN {X 0,Y 245.117,Z 841.277,A -85,B 0,C 180,E1 -25516.74,E2 -25516.74} C_VEL
LIN {X 0,Y 254.736,Z 826.348,A -85,B 0,C 180,E1 -25519.944,E2 -25519.944} C_VEL
LIN {X 0,Y 264.011,Z 810.344,A -85,B 0,C 180,E1 -25522.687,E2 -25522.687} C_VEL
LIN {X 0,Y 272.725,Z 793.383,A -85,B 0,C 180,E1 -25525.026,E2 -25525.026} C_VEL
LIN {X 0,Y 280.716,Z 775.526,A -85,B 0,C 180,E1 -25527.017,E2 -25527.017} C_VEL
LIN {X 0,Y 287.85,Z 756.807,A -85,B 0,C 180,E1 -25528.706,E2 -25528.706} C_VEL
LIN {X 0,Y 294.047,Z 737.187,A -85,B 0,C 180,E1 -25530.125,E2 -25530.125} C_VEL
LIN {X 0,Y 299.024,Z 717.296,A -85,B 0,C 180,E1 -25531.273,E2 -25531.273} C_VEL
LIN {X 0,Y 306.803,Z 679.572,A -85,B 0,C 180,E1 -25532.954,E2 -25532.954} C_VEL
LIN {X 0,Y 314.485,Z 640.094,A -85,B 0,C 180,E1 -25534.3,E2 -25534.3} C_VEL
LIN {X 0,Y 322.291,Z 594.861,A -85,B 0,C 180,E1 -25535.463,E2 -25535.463} C_VEL
LIN {X 0,Y 328.535,Z 550.082,A -85,B 0,C 180,E1 -25536.422,E2 -25536.422} C_VEL
LIN {X 0,Y 334.258,Z 494.763,A -85,B 0,C 180,E1 -25537.414,E2 -25537.414} C_VEL
LIN {X 0,Y 336.896,Z 469.242,A -85,B 0,C 180,E1 -25537.856,E2 -25537.856} C_VEL
LIN {X 0,Y 340.426,Z 454.288,A -85,B 0,C 180,E1 -25538.279,E2 -25538.279} C_VEL
LIN {X 0,Y 338.052,Z 443.9,A -85,B 0,C 180,E1 -25541.281,E2 -25541.281} C_VEL
LIN {X 0,Y 335.855,Z 434.787,A -85,B 0,C 180,E1 -25544.502,E2 -25544.502} C_VEL
LIN {X 0,Y 334.307,Z 428.715,A -85,B 0,C 180,E1 -25547.159,E2 -25547.159} C_VEL
LIN {X 0,Y 333.429,Z 427.235,A -85,B 0,C 180,E1 -25548.458,E2 -25548.458} C_VEL
LIN {X 0,Y 331.509,Z 427.281,A -85,B 0,C 180,E1 -25550.847,E2 -25550.847} C_VEL
LIN {X 0,Y 330.247,Z 427.072,A -85,B 0,C 180,E1 -25552.881,E2 -25552.881} C_VEL
LIN {X 0,Y 330.126,Z 426.75,A -85,B 0,C 180,E1 -25553.266,E2 -25553.266} C_VEL
LIN {X 0,Y 329.901,Z 423.004,A -85,B 0,C 180,E1 -25557.394,E2 -25557.394} C_VEL
LIN {X 0,Y 330.781,Z 422.255,A -85,B 0,C 180,E1 -25562.252,E2 -25562.252} C_VEL
LIN {X 0,Y 331.614,Z 422.963,A -85,B 0,C 180,E1 -25564.496,E2 -25564.496} C_VEL
LIN {X 0,Y 332.18,Z 436.644,A -85,B 0,C 180,E1 -25569.005,E2 -25569.005} C_VEL
LIN {X 0,Y 334.634,Z 454.529,A -85,B 0,C 180,E1 -25573.915,E2 -25573.915} C_VEL
LIN {X 0,Y 317.576,Z 549.187,A -85,B 0,C 180,E1 -25576.291,E2 -25576.291} C_VEL
LIN {X 0,Y 311.251,Z 614.325,A -85,B 0,C 180,E1 -25577.655,E2 -25577.655} C_VEL
LIN {X 0,Y 305.933,Z 651.501,A -85,B 0,C 180,E1 -25578.497,E2 -25578.497} C_VEL
LIN {X 0,Y 299.223,Z 687.667,A -85,B 0,C 180,E1 -25579.552,E2 -25579.552} C_VEL
LIN {X 0,Y 291.639,Z 721.28,A -85,B 0,C 180,E1 -25580.771,E2 -25580.771} C_VEL
LIN {X 0,Y 283.713,Z 752.096,A -85,B 0,C 180,E1 -25582.179,E2 -25582.179} C_VEL
LIN {X 0,Y 275.126,Z 782.04,A -85,B 0,C 180,E1 -25583.936,E2 -25583.936} C_VEL
LIN {X 0,Y 268.417,Z 801.547,A -85,B 0,C 180,E1 -25585.366,E2 -25585.366} C_VEL
LIN {X 0,Y 260.644,Z 820.526,A -85,B 0,C 180,E1 -25587.126,E2 -25587.126} C_VEL
LIN {X 0,Y 252.122,Z 838.586,A -85,B 0,C 180,E1 -25589.25,E2 -25589.25} C_VEL
LIN {X 0,Y 243.257,Z 855.197,A -85,B 0,C 180,E1 -25591.695,E2 -25591.695} C_VEL
LIN {X 0,Y 233.594,Z 871.554,A -85,B 0,C 180,E1 -25594.73,E2 -25594.73} C_VEL
LIN {X 0,Y 224.091,Z 886.437,A -85,B 0,C 180,E1 -25598.251,E2 -25598.251} C_VEL
LIN {X 0,Y 214.948,Z 899.902,A -85,B 0,C 180,E1 -25602.3,E2 -25602.3} C_VEL
LIN {X 0,Y 206.322,Z 912.249,A -85,B 0,C 180,E1 -25607.037,E2 -25607.037} C_VEL
LIN {X 0,Y 198.346,Z 923.808,A -85,B 0,C 180,E1 -25612.776,E2 -25612.776} C_VEL
LIN {X 0,Y 192.471,Z 932.966,A -85,B 0,C 180,E1 -25618.701,E2 -25618.701} C_VEL
LIN {X 0,Y 188.332,Z 940.658,A -85,B 0,C 180,E1 -25625.213,E2 -25625.213} C_VEL
LIN {X 0,Y 186.215,Z 946.456,A -85,B 0,C 180,E1 -25631.882,E2 -25631.882} C_VEL
LIN {X 0,Y 185.881,Z 950.495,A -85,B 0,C 180,E1 -25638.52,E2 -25638.52} C_VEL
LIN {X 0,Y 186.572,Z 952.702,A -85,B 0,C 180,E1 -25644.464,E2 -25644.464} C_VEL
LIN {X 0,Y 187.122,Z 953.372,A -85,B 0,C 180,E1 -25648.775,E2 -25648.775} C_VEL
LIN {X 0,Y 187.016,Z 953.251,A -85,B 0,C 180,E1 -25652.758,E2 -25652.758} C_VEL
LIN {X 0,Y 186.372,Z 951.942,A -85,B 0,C 180,E1 -25658.019,E2 -25658.019} C_VEL
LIN {X 0,Y 186.121,Z 950.581,A -85,B 0,C 180,E1 -25661.78,E2 -25661.78} C_VEL
LIN {X 0,Y 186.54,Z 950.022,A -85,B 0,C 180,E1 -25669.411,E2 -25669.411} C_VEL
LIN {X 0,Y 190.211,Z 947.854,A -85,B 0,C 180,E1 -25677.895,E2 -25677.895} C_VEL
LIN {X 0,Y 200.211,Z 943.1,A -85,B 0,C 180,E1 -25687.9,E2 -25687.9} C_VEL
LIN {X 0,Y 215.395,Z 936.848,A -85,B 0,C 180,E1 -25696.4,E2 -25696.4} C_VEL
LIN {X 0,Y 235.218,Z 929.227,A -85,B 0,C 180,E1 -25703.478,E2 -25703.478} C_VEL
LIN {X 0,Y 220.878,Z 928.989,A -85,B 0,C 180,E1 -25708.324,E2 -25708.324} C_VEL
LIN {X 0,Y 208.835,Z 927.095,A -85,B 0,C 180,E1 -25713.865,E2 -25713.865} C_VEL
LIN {X 0,Y 200.03,Z 923.715,A -85,B 0,C 180,E1 -25719.518,E2 -25719.518} C_VEL
LIN {X 0,Y 193.497,Z 918.5,A -85,B 0,C 180,E1 -25725.638,E2 -25725.638} C_VEL
LIN {X 0,Y 189.37,Z 911.663,A -85,B 0,C 180,E1 -25731.804,E2 -25731.804} C_VEL
LIN {X 0,Y 187.278,Z 903.762,A -85,B 0,C 180,E1 -25737.552,E2 -25737.552} C_VEL
LIN {X 0,Y 186.475,Z 894.015,A -85,B 0,C 180,E1 -25743.381,E2 -25743.381} C_VEL
LIN {X 0,Y 186.765,Z 882.809,A -85,B 0,C 180,E1 -25748.932,E2 -25748.932} C_VEL
LIN {X 0,Y 187.99,Z 870.181,A -85,B 0,C 180,E1 -25754.162,E2 -25754.162} C_VEL
LIN {X 0,Y 190.271,Z 855.222,A -85,B 0,C 180,E1 -25759.334,E2 -25759.334} C_VEL
LIN {X 0,Y 190.434,Z 854.584,A -85,B 0,C 180,E1 -25759.636,E2 -25759.636} C_VEL
LIN {X 0,Y 191.918,Z 854.122,A -85,B 0,C 180,E1 -25761.069,E2 -25761.069} C_VEL
LIN {X 0,Y 194.691,Z 852.79,A -85,B 0,C 180,E1 -25762.655,E2 -25762.655} C_VEL
LIN {X 0,Y 197.716,Z 851.58,A -85,B 0,C 180,E1 -25764.5,E2 -25764.5} C_VEL
LIN {X 0,Y 199.738,Z 850.686,A -85,B 0,C 180,E1 -25765.5,E2 -25765.5} C_VEL
LIN {X 0,Y 203.867,Z 849.004,A -85,B 0,C 180,E1 -25767.454,E2 -25767.454} C_VEL
LIN {X 0,Y 210.165,Z 846.505,A -85,B 0,C 180,E1 -25770.015,E2 -25770.015} C_VEL
LIN {X 0,Y 217.554,Z 843.54,A -85,B 0,C 180,E1 -25772.53,E2 -25772.53} C_VEL
LIN {X 0,Y 225.682,Z 840.264,A -85,B 0,C 180,E1 -25774.858,E2 -25774.858} C_VEL
LIN {X 0,Y 235.195,Z 836.31,A -85,B 0,C 180,E1 -25777.135,E2 -25777.135} C_VEL
LIN {X 0,Y 246.225,Z 831.487,A -85,B 0,C 180,E1 -25779.309,E2 -25779.309} C_VEL
LIN {X 0,Y 247.205,Z 831.074,A -85,B 0,C 180,E1 -25779.498,E2 -25779.498} C_VEL
LIN {X 0,Y 237.234,Z 845.705,A -85,B 0,C 180,E1 -25782.83,E2 -25782.83} C_VEL
LIN {X 0,Y 227.334,Z 858.969,A -85,B 0,C 180,E1 -25786.674,E2 -25786.674} C_VEL
LIN {X 0,Y 217.886,Z 870.69,A -85,B 0,C 180,E1 -25791.045,E2 -25791.045} C_VEL
LIN {X 0,Y 209.2,Z 880.866,A -85,B 0,C 180,E1 -25795.998,E2 -25795.998} C_VEL
LIN {X 0,Y 201.59,Z 889.464,A -85,B 0,C 180,E1 -25801.565,E2 -25801.565} C_VEL
LIN {X 0,Y 195.631,Z 896.147,A -85,B 0,C 180,E1 -25807.459,E2 -25807.459} C_VEL
LIN {X 0,Y 191.358,Z 901.064,A -85,B 0,C 180,E1 -25813.61,E2 -25813.61} C_VEL
LIN {X 0,Y 188.707,Z 904.318,A -85,B 0,C 180,E1 -25819.93,E2 -25819.93} C_VEL
LIN {X 0,Y 187.458,Z 905.963,A -85,B 0,C 180,E1 -25826.33,E2 -25826.33} C_VEL
LIN {X 0,Y 187.348,Z 906.093,A -85,B 0,C 180,E1 -25832.447,E2 -25832.447} C_VEL
LIN {X 0,Y 188.268,Z 904.854,A -85,B 0,C 180,E1 -25838.552,E2 -25838.552} C_VEL
LIN {X 0,Y 190.688,Z 901.864,A -85,B 0,C 180,E1 -25845.199,E2 -25845.199} C_VEL
LIN {X 0,Y 194.864,Z 897.067,A -85,B 0,C 180,E1 -25851.681,E2 -25851.681} C_VEL
LIN {X 0,Y 200.552,Z 890.69,A -85,B 0,C 180,E1 -25857.624,E2 -25857.624} C_VEL
LIN {X 0,Y 207.917,Z 882.411,A -85,B 0,C 180,E1 -25863.246,E2 -25863.246} C_VEL
LIN {X 0,Y 216.245,Z 872.748,A -85,B 0,C 180,E1 -25868.181,E2 -25868.181} C_VEL
LIN {X 0,Y 225.396,Z 861.565,A -85,B 0,C 180,E1 -25872.574,E2 -25872.574} C_VEL
LIN {X 0,Y 234.952,Z 849.037,A -85,B 0,C 180,E1 -25876.415,E2 -25876.415} C_VEL
LIN {X 0,Y 244.778,Z 835.009,A -85,B 0,C 180,E1 -25879.807,E2 -25879.807} C_VEL
LIN {X 0,Y 254.613,Z 819.47,A -85,B 0,C 180,E1 -25882.787,E2 -25882.787} C_VEL
LIN {X 0,Y 263.892,Z 803.012,A -85,B 0,C 180,E1 -25885.307,E2 -25885.307} C_VEL
LIN {X 0,Y 272.434,Z 785.735,A -85,B 0,C 180,E1 -25887.437,E2 -25887.437} C_VEL
LIN {X 0,Y 279.957,Z 768.107,A -85,B 0,C 180,E1 -25889.201,E2 -25889.201} C_VEL
LIN {X 0,Y 286.635,Z 749.617,A -85,B 0,C 180,E1 -25890.703,E2 -25890.703} C_VEL
LIN {X 0,Y 292.294,Z 730.504,A -85,B 0,C 180,E1 -25891.954,E2 -25891.954} C_VEL
LIN {X 0,Y 297.469,Z 708.123,A -85,B 0,C 180,E1 -25893.114,E2 -25893.114} C_VEL
LIN {X 0,Y 305.494,Z 669.757,A -85,B 0,C 180,E1 -25894.698,E2 -25894.698} C_VEL
LIN {X 0,Y 313.232,Z 629.98,A -85,B 0,C 180,E1 -25895.932,E2 -25895.932} C_VEL
LIN {X 0,Y 320.771,Z 585.376,A -85,B 0,C 180,E1 -25897.004,E2 -25897.004} C_VEL
LIN {X 0,Y 326.845,Z 539.857,A -85,B 0,C 180,E1 -25897.922,E2 -25897.922} C_VEL
LIN {X 0,Y 333.775,Z 472.082,A -85,B 0,C 180,E1 -25899.089,E2 -25899.089} C_VEL
LIN {X 0,Y 336.956,Z 458.646,A -85,B 0,C 180,E1 -25899.457,E2 -25899.457} C_VEL
LIN {X 0,Y 334.834,Z 448.807,A -85,B 0,C 180,E1 -25902.446,E2 -25902.446} C_VEL
LIN {X 0,Y 333.061,Z 440.864,A -85,B 0,C 180,E1 -25905.393,E2 -25905.393} C_VEL
LIN {X 0,Y 331.576,Z 434.33,A -85,B 0,C 180,E1 -25908.432,E2 -25908.432} C_VEL
LIN {X 0,Y 330.555,Z 429.261,A -85,B 0,C 180,E1 -25911.476,E2 -25911.476} C_VEL
LIN {X 0,Y 330.126,Z 426.75,A -85,B 0,C 180,E1 -25913.266,E2 -25913.266} C_VEL
LIN {X 0,Y 329.666,Z 426.429,A -85,B 0,C 180,E1 -25914.614,E2 -25914.614} C_VEL
LIN {X 0,Y 328.616,Z 428.738,A -85,B 0,C 180,E1 -25917.021,E2 -25917.021} C_VEL
LIN {X 0,Y 328.152,Z 430.31,A -85,B 0,C 180,E1 -25918.971,E2 -25918.971} C_VEL
LIN {X 0,Y 328.183,Z 430.311,A -85,B 0,C 180,E1 -25919.463,E2 -25919.463} C_VEL
LIN {X 0,Y 329.15,Z 430.15,A -85,B 0,C 180,E1 -25922.96,E2 -25922.96} C_VEL
LIN {X 0,Y 329.646,Z 430.754,A -85,B 0,C 180,E1 -25924.218,E2 -25924.218} C_VEL
LIN {X 0,Y 330.058,Z 443.709,A -85,B 0,C 180,E1 -25928.449,E2 -25928.449} C_VEL
LIN {X 0,Y 331.816,Z 458.871,A -85,B 0,C 180,E1 -25932.675,E2 -25932.675} C_VEL
LIN {X 0,Y 315.61,Z 546.131,A -85,B 0,C 180,E1 -25934.834,E2 -25934.834} C_VEL
LIN {X 0,Y 309.065,Z 611.623,A -85,B 0,C 180,E1 -25936.188,E2 -25936.188} C_VEL
LIN {X 0,Y 303.553,Z 649.408,A -85,B 0,C 180,E1 -25937.026,E2 -25937.026} C_VEL
LIN {X 0,Y 296.75,Z 685.329,A -85,B 0,C 180,E1 -25938.043,E2 -25938.043} C_VEL
LIN {X 0,Y 289.056,Z 718.97,A -85,B 0,C 180,E1 -25939.223,E2 -25939.223} C_VEL
LIN {X 0,Y 280.917,Z 750.037,A -85,B 0,C 180,E1 -25940.591,E2 -25940.591} C_VEL
LIN {X 0,Y 271.892,Z 780.773,A -85,B 0,C 180,E1 -25942.347,E2 -25942.347} C_VEL
LIN {X 0,Y 264.922,Z 800.426,A -85,B 0,C 180,E1 -25943.757,E2 -25943.757} C_VEL
LIN {X 0,Y 256.966,Z 819.279,A -85,B 0,C 180,E1 -25945.479,E2 -25945.479} C_VEL
LIN {X 0,Y 248.159,Z 837.343,A -85,B 0,C 180,E1 -25947.572,E2 -25947.572} C_VEL
LIN {X 0,Y 238.952,Z 853.946,A -85,B 0,C 180,E1 -25949.981,E2 -25949.981} C_VEL
LIN {X 0,Y 228.906,Z 870.34,A -85,B 0,C 180,E1 -25952.999,E2 -25952.999} C_VEL
LIN {X 0,Y 218.97,Z 885.214,A -85,B 0,C 180,E1 -25956.518,E2 -25956.518} C_VEL
LIN {X 0,Y 209.353,Z 898.701,A -85,B 0,C 180,E1 -25960.589,E2 -25960.589} C_VEL
LIN {X 0,Y 200.403,Z 910.85,A -85,B 0,C 180,E1 -25965.291,E2 -25965.291} C_VEL
LIN {X 0,Y 192.068,Z 922.146,A -85,B 0,C 180,E1 -25970.956,E2 -25970.956} C_VEL
LIN {X 0,Y 185.619,Z 931.433,A -85,B 0,C 180,E1 -25977.039,E2 -25977.039} C_VEL
LIN {X 0,Y 180.96,Z 939.232,A -85,B 0,C 180,E1 -25983.766,E2 -25983.766} C_VEL
LIN {X 0,Y 178.449,Z 945.149,A -85,B 0,C 180,E1 -25990.696,E2 -25990.696} C_VEL
LIN {X 0,Y 177.881,Z 949.309,A -85,B 0,C 180,E1 -25997.667,E2 -25997.667} C_VEL
LIN {X 0,Y 178.527,Z 951.616,A -85,B 0,C 180,E1 -26003.892,E2 -26003.892} C_VEL
LIN {X 0,Y 179.15,Z 952.346,A -85,B 0,C 180,E1 -26008.401,E2 -26008.401} C_VEL
LIN {X 0,Y 179.119,Z 952.298,A -85,B 0,C 180,E1 -26012.248,E2 -26012.248} C_VEL
LIN {X 0,Y 178.478,Z 951.231,A -85,B 0,C 180,E1 -26017.425,E2 -26017.425} C_VEL
LIN {X 0,Y 178.201,Z 948.82,A -85,B 0,C 180,E1 -26023.901,E2 -26023.901} C_VEL
LIN {X 0,Y 179.565,Z 948.028,A -85,B 0,C 180,E1 -26032.596,E2 -26032.596} C_VEL
LIN {X 0,Y 184.909,Z 945.615,A -85,B 0,C 180,E1 -26041.637,E2 -26041.637} C_VEL
LIN {X 0,Y 198.035,Z 940.497,A -85,B 0,C 180,E1 -26052.185,E2 -26052.185} C_VEL
LIN {X 0,Y 215.595,Z 934.277,A -85,B 0,C 180,E1 -26060.343,E2 -26060.343} C_VEL
LIN {X 0,Y 224.946,Z 931.062,A -85,B 0,C 180,E1 -26063.521,E2 -26063.521} C_VEL
LIN {X 0,Y 210.323,Z 929.897,A -85,B 0,C 180,E1 -26068.789,E2 -26068.789} C_VEL
LIN {X 0,Y 199.011,Z 927.195,A -85,B 0,C 180,E1 -26074.4,E2 -26074.4} C_VEL
LIN {X 0,Y 190.144,Z 922.711,A -85,B 0,C 180,E1 -26080.653,E2 -26080.653} C_VEL
LIN {X 0,Y 184.091,Z 916.502,A -85,B 0,C 180,E1 -26087.133,E2 -26087.133} C_VEL
LIN {X 0,Y 180.604,Z 909.093,A -85,B 0,C 180,E1 -26093.323,E2 -26093.323} C_VEL
LIN {X 0,Y 178.898,Z 900.333,A -85,B 0,C 180,E1 -26099.36,E2 -26099.36} C_VEL
LIN {X 0,Y 178.467,Z 890.241,A -85,B 0,C 180,E1 -26105.143,E2 -26105.143} C_VEL
LIN {X 0,Y 179.045,Z 878.857,A -85,B 0,C 180,E1 -26110.62,E2 -26110.62} C_VEL
LIN {X 0,Y 180.645,Z 865.331,A -85,B 0,C 180,E1 -26116.067,E2 -26116.067} C_VEL
LIN {X 0,Y 181.259,Z 861.357,A -85,B 0,C 180,E1 -26117.496,E2 -26117.496} C_VEL
LIN {X 0,Y 182.655,Z 860.881,A -85,B 0,C 180,E1 -26119.175,E2 -26119.175} C_VEL
LIN {X 0,Y 184.878,Z 859.719,A -85,B 0,C 180,E1 -26120.582,E2 -26120.582} C_VEL
LIN {X 0,Y 187.455,Z 858.737,A -85,B 0,C 180,E1 -26122.585,E2 -26122.585} C_VEL
LIN {X 0,Y 189.402,Z 857.837,A -85,B 0,C 180,E1 -26123.655,E2 -26123.655} C_VEL
LIN {X 0,Y 193.084,Z 856.41,A -85,B 0,C 180,E1 -26125.785,E2 -26125.785} C_VEL
LIN {X 0,Y 199.5,Z 853.891,A -85,B 0,C 180,E1 -26128.761,E2 -26128.761} C_VEL
LIN {X 0,Y 205.998,Z 851.449,A -85,B 0,C 180,E1 -26131.319,E2 -26131.319} C_VEL
LIN {X 0,Y 213.66,Z 848.533,A -85,B 0,C 180,E1 -26133.842,E2 -26133.842} C_VEL
LIN {X 0,Y 222.793,Z 845.011,A -85,B 0,C 180,E1 -26136.329,E2 -26136.329} C_VEL
LIN {X 0,Y 232.579,Z 841.124,A -85,B 0,C 180,E1 -26138.563,E2 -26138.563} C_VEL
LIN {X 0,Y 237.354,Z 839.232,A -85,B 0,C 180,E1 -26139.563,E2 -26139.563} C_VEL
LIN {X 0,Y 227.209,Z 852.939,A -85,B 0,C 180,E1 -26143.069,E2 -26143.069} C_VEL
LIN {X 0,Y 217.313,Z 865.212,A -85,B 0,C 180,E1 -26147.08,E2 -26147.08} C_VEL
LIN {X 0,Y 207.93,Z 876.049,A -85,B 0,C 180,E1 -26151.659,E2 -26151.659} C_VEL
LIN {X 0,Y 199.311,Z 885.495,A -85,B 0,C 180,E1 -26156.908,E2 -26156.908} C_VEL
LIN {X 0,Y 191.988,Z 893.271,A -85,B 0,C 180,E1 -26162.722,E2 -26162.722} C_VEL
LIN {X 0,Y 186.123,Z 899.5,A -85,B 0,C 180,E1 -26169.233,E2 -26169.233} C_VEL
LIN {X 0,Y 182.16,Z 903.835,A -85,B 0,C 180,E1 -26176.024,E2 -26176.024} C_VEL
LIN {X 0,Y 180.068,Z 906.292,A -85,B 0,C 180,E1 -26182.662,E2 -26182.662} C_VEL
LIN {X 0,Y 179.346,Z 907.18,A -85,B 0,C 180,E1 -26189.041,E2 -26189.041} C_VEL
LIN {X 0,Y 179.713,Z 906.706,A -85,B 0,C 180,E1 -26195.427,E2 -26195.427} C_VEL
LIN {X 0,Y 181.37,Z 904.722,A -85,B 0,C 180,E1 -26202.092,E2 -26202.092} C_VEL
LIN {X 0,Y 184.599,Z 901.148,A -85,B 0,C 180,E1 -26208.637,E2 -26208.637} C_VEL
LIN {X 0,Y 189.559,Z 895.888,A -85,B 0,C 180,E1 -26214.96,E2 -26214.96} C_VEL
LIN {X 0,Y 195.918,Z 889.209,A -85,B 0,C 180,E1 -26220.688,E2 -26220.688} C_VEL
LIN {X 0,Y 203.809,Z 880.749,A -85,B 0,C 180,E1 -26226.066,E2 -26226.066} C_VEL
LIN {X 0,Y 212.618,Z 870.897,A -85,B 0,C 180,E1 -26230.82,E2 -26230.82} C_VEL
LIN {X 0,Y 222.139,Z 859.575,A -85,B 0,C 180,E1 -26235.034,E2 -26235.034} C_VEL
LIN {X 0,Y 232.373,Z 846.387,A -85,B 0,C 180,E1 -26238.852,E2 -26238.852} C_VEL
LIN {X 0,Y 242.393,Z 832.229,A -85,B 0,C 180,E1 -26242.074,E2 -26242.074} C_VEL
LIN {X 0,Y 252.019,Z 817.122,A -85,B 0,C 180,E1 -26244.816,E2 -26244.816} C_VEL
LIN {X 0,Y 261.527,Z 800.292,A -85,B 0,C 180,E1 -26247.259,E2 -26247.259} C_VEL
LIN {X 0,Y 270.277,Z 782.497,A -85,B 0,C 180,E1 -26249.331,E2 -26249.331} C_VEL
LIN {X 0,Y 277.78,Z 764.721,A -85,B 0,C 180,E1 -26251.009,E2 -26251.009} C_VEL
LIN {X 0,Y 284.302,Z 746.388,A -85,B 0,C 180,E1 -26252.41,E2 -26252.41} C_VEL
LIN {X 0,Y 290.104,Z 726.061,A -85,B 0,C 180,E1 -26253.654,E2 -26253.654} C_VEL
LIN {X 0,Y 298.349,Z 689.251,A -85,B 0,C 180,E1 -26255.363,E2 -26255.363} C_VEL
LIN {X 0,Y 306.571,Z 649.532,A -85,B 0,C 180,E1 -26256.763,E2 -26256.763} C_VEL
LIN {X 0,Y 314.849,Z 604.958,A -85,B 0,C 180,E1 -26257.916,E2 -26257.916} C_VEL
LIN {X 0,Y 321.643,Z 559.448,A -85,B 0,C 180,E1 -26258.879,E2 -26258.879} C_VEL
LIN {X 0,Y 326.934,Z 512.22,A -85,B 0,C 180,E1 -26259.721,E2 -26259.721} C_VEL
LIN {X 0,Y 330.832,Z 474.84,A -85,B 0,C 180,E1 -26260.347,E2 -26260.347} C_VEL
LIN {X 0,Y 333.615,Z 463.08,A -85,B 0,C 180,E1 -26260.659,E2 -26260.659} C_VEL
LIN {X 0,Y 331.652,Z 453.139,A -85,B 0,C 180,E1 -26263.852,E2 -26263.852} C_VEL
LIN {X 0,Y 330.07,Z 445.457,A -85,B 0,C 180,E1 -26266.957,E2 -26266.957} C_VEL
LIN {X 0,Y 328.824,Z 439.214,A -85,B 0,C 180,E1 -26270.196,E2 -26270.196} C_VEL
LIN {X 0,Y 328.084,Z 434.344,A -85,B 0,C 180,E1 -26273.525,E2 -26273.525} C_VEL
LIN {X 0,Y 328.08,Z 430.764,A -85,B 0,C 180,E1 -26277.555,E2 -26277.555} C_VEL
LIN {X 0,Y 328.183,Z 430.311,A -85,B 0,C 180,E1 -26279.463,E2 -26279.463} C_VEL
LIN {X 0,Y 328.234,Z 430.925,A -85,B 0,C 180,E1 -26280.722,E2 -26280.722} C_VEL
LIN {X 0,Y 328.04,Z 433.786,A -85,B 0,C 180,E1 -26282.307,E2 -26282.307} C_VEL
LIN {X 0,Y 327.611,Z 441.652,A -85,B 0,C 180,E1 -26284.981,E2 -26284.981} C_VEL
LIN {X 0,Y 327.603,Z 442.751,A -85,B 0,C 180,E1 -26285.334,E2 -26285.334} C_VEL
LIN {X 0,Y 327.955,Z 451.516,A -85,B 0,C 180,E1 -26288.106,E2 -26288.106} C_VEL
LIN {X 0,Y 329.07,Z 463.463,A -85,B 0,C 180,E1 -26291.433,E2 -26291.433} C_VEL
LIN {X 0,Y 313.808,Z 543.454,A -85,B 0,C 180,E1 -26293.365,E2 -26293.365} C_VEL
LIN {X 0,Y 307.081,Z 608.92,A -85,B 0,C 180,E1 -26294.7,E2 -26294.7} C_VEL
LIN {X 0,Y 301.411,Z 647.092,A -85,B 0,C 180,E1 -26295.528,E2 -26295.528} C_VEL
LIN {X 0,Y 294.353,Z 683.739,A -85,B 0,C 180,E1 -26296.532,E2 -26296.532} C_VEL
LIN {X 0,Y 286.597,Z 716.892,A -85,B 0,C 180,E1 -26297.657,E2 -26297.657} C_VEL
LIN {X 0,Y 278.138,Z 748.638,A -85,B 0,C 180,E1 -26299.009,E2 -26299.009} C_VEL
LIN {X 0,Y 268.869,Z 779.544,A -85,B 0,C 180,E1 -26300.724,E2 -26300.724} C_VEL
LIN {X 0,Y 261.589,Z 799.487,A -85,B 0,C 180,E1 -26302.121,E2 -26302.121} C_VEL
LIN {X 0,Y 253.148,Z 818.845,A -85,B 0,C 180,E1 -26303.865,E2 -26303.865} C_VEL
LIN {X 0,Y 244.04,Z 836.835,A -85,B 0,C 180,E1 -26305.928,E2 -26305.928} C_VEL
LIN {X 0,Y 234.164,Z 853.928,A -85,B 0,C 180,E1 -26308.403,E2 -26308.403} C_VEL
LIN {X 0,Y 223.428,Z 870.565,A -85,B 0,C 180,E1 -26311.512,E2 -26311.512} C_VEL
LIN {X 0,Y 212.82,Z 885.678,A -85,B 0,C 180,E1 -26315.165,E2 -26315.165} C_VEL
LIN {X 0,Y 202.292,Z 899.686,A -85,B 0,C 180,E1 -26319.55,E2 -26319.55} C_VEL
LIN {X 0,Y 192.565,Z 912.154,A -85,B 0,C 180,E1 -26324.654,E2 -26324.654} C_VEL
LIN {X 0,Y 184.042,Z 923.07,A -85,B 0,C 180,E1 -26330.532,E2 -26330.532} C_VEL
LIN {X 0,Y 177.196,Z 932.344,A -85,B 0,C 180,E1 -26337.2,E2 -26337.2} C_VEL
LIN {X 0,Y 172.463,Z 939.992,A -85,B 0,C 180,E1 -26344.594,E2 -26344.594} C_VEL
LIN {X 0,Y 170.238,Z 945.439,A -85,B 0,C 180,E1 -26351.863,E2 -26351.863} C_VEL
LIN {X 0,Y 169.969,Z 949.01,A -85,B 0,C 180,E1 -26358.806,E2 -26358.806} C_VEL
LIN {X 0,Y 170.741,Z 950.877,A -85,B 0,C 180,E1 -26364.961,E2 -26364.961} C_VEL
LIN {X 0,Y 171.274,Z 951.411,A -85,B 0,C 180,E1 -26369.331,E2 -26369.331} C_VEL
LIN {X 0,Y 171.013,Z 951.145,A -85,B 0,C 180,E1 -26373.688,E2 -26373.688} C_VEL
LIN {X 0,Y 170.316,Z 949.666,A -85,B 0,C 180,E1 -26379.495,E2 -26379.495} C_VEL
LIN {X 0,Y 170.453,Z 946.959,A -85,B 0,C 180,E1 -26386.004,E2 -26386.004} C_VEL
LIN {X 0,Y 173.084,Z 945.951,A -85,B 0,C 180,E1 -26396.043,E2 -26396.043} C_VEL
LIN {X 0,Y 180.438,Z 943.331,A -85,B 0,C 180,E1 -26405.581,E2 -26405.581} C_VEL
LIN {X 0,Y 196.51,Z 938.088,A -85,B 0,C 180,E1 -26416.264,E2 -26416.264} C_VEL
LIN {X 0,Y 214.673,Z 932.431,A -85,B 0,C 180,E1 -26423.559,E2 -26423.559} C_VEL
LIN {X 0,Y 200.309,Z 930.401,A -85,B 0,C 180,E1 -26429.059,E2 -26429.059} C_VEL
LIN {X 0,Y 189.197,Z 926.855,A -85,B 0,C 180,E1 -26434.989,E2 -26434.989} C_VEL
LIN {X 0,Y 180.649,Z 921.423,A -85,B 0,C 180,E1 -26441.609,E2 -26441.609} C_VEL
LIN {X 0,Y 175.206,Z 914.675,A -85,B 0,C 180,E1 -26448.144,E2 -26448.144} C_VEL
LIN {X 0,Y 171.943,Z 906.056,A -85,B 0,C 180,E1 -26454.996,E2 -26454.996} C_VEL
LIN {X 0,Y 170.634,Z 896.398,A -85,B 0,C 180,E1 -26461.343,E2 -26461.343} C_VEL
LIN {X 0,Y 170.574,Z 886.025,A -85,B 0,C 180,E1 -26467.071,E2 -26467.071} C_VEL
LIN {X 0,Y 171.537,Z 873.666,A -85,B 0,C 180,E1 -26472.797,E2 -26472.797} C_VEL
LIN {X 0,Y 172.27,Z 867.893,A -85,B 0,C 180,E1 -26475.199,E2 -26475.199} C_VEL
LIN {X 0,Y 173.563,Z 867.342,A -85,B 0,C 180,E1 -26477.086,E2 -26477.086} C_VEL
LIN {X 0,Y 175.531,Z 866.293,A -85,B 0,C 180,E1 -26478.602,E2 -26478.602} C_VEL
LIN {X 0,Y 177.882,Z 865.321,A -85,B 0,C 180,E1 -26480.74,E2 -26480.74} C_VEL
LIN {X 0,Y 179.964,Z 864.415,A -85,B 0,C 180,E1 -26482.198,E2 -26482.198} C_VEL
LIN {X 0,Y 188.449,Z 861.09,A -85,B 0,C 180,E1 -26487.149,E2 -26487.149} C_VEL
LIN {X 0,Y 195.136,Z 858.622,A -85,B 0,C 180,E1 -26490.143,E2 -26490.143} C_VEL
LIN {X 0,Y 201.808,Z 856.237,A -85,B 0,C 180,E1 -26492.688,E2 -26492.688} C_VEL
LIN {X 0,Y 210.529,Z 853.073,A -85,B 0,C 180,E1 -26495.411,E2 -26495.411} C_VEL
LIN {X 0,Y 219.938,Z 849.575,A -85,B 0,C 180,E1 -26497.861,E2 -26497.861} C_VEL
LIN {X 0,Y 227.467,Z 846.873,A -85,B 0,C 180,E1 -26499.623,E2 -26499.623} C_VEL
LIN {X 0,Y 216.58,Z 860.42,A -85,B 0,C 180,E1 -26503.545,E2 -26503.545} C_VEL
LIN {X 0,Y 206.231,Z 872.237,A -85,B 0,C 180,E1 -26508.004,E2 -26508.004} C_VEL
LIN {X 0,Y 196.607,Z 882.512,A -85,B 0,C 180,E1 -26513.122,E2 -26513.122} C_VEL
LIN {X 0,Y 188.064,Z 891.201,A -85,B 0,C 180,E1 -26518.954,E2 -26518.954} C_VEL
LIN {X 0,Y 180.987,Z 898.208,A -85,B 0,C 180,E1 -26525.521,E2 -26525.521} C_VEL
LIN {X 0,Y 176.12,Z 903.1,A -85,B 0,C 180,E1 -26532.147,E2 -26532.147} C_VEL
LIN {X 0,Y 172.956,Z 906.436,A -85,B 0,C 180,E1 -26539.339,E2 -26539.339} C_VEL
LIN {X 0,Y 171.582,Z 908.023,A -85,B 0,C 180,E1 -26546.324,E2 -26546.324} C_VEL
LIN {X 0,Y 171.513,Z 908.078,A -85,B 0,C 180,E1 -26553.007,E2 -26553.007} C_VEL
LIN {X 0,Y 172.643,Z 906.767,A -85,B 0,C 180,E1 -26559.669,E2 -26559.669} C_VEL
LIN {X 0,Y 175.352,Z 903.885,A -85,B 0,C 180,E1 -26566.565,E2 -26566.565} C_VEL
LIN {X 0,Y 179.86,Z 899.366,A -85,B 0,C 180,E1 -26573.248,E2 -26573.248} C_VEL
LIN {X 0,Y 186.196,Z 893.1,A -85,B 0,C 180,E1 -26579.607,E2 -26579.607} C_VEL
LIN {X 0,Y 194.323,Z 884.947,A -85,B 0,C 180,E1 -26585.552,E2 -26585.552} C_VEL
LIN {X 0,Y 203.592,Z 875.25,A -85,B 0,C 180,E1 -26590.783,E2 -26590.783} C_VEL
LIN {X 0,Y 213.642,Z 864.047,A -85,B 0,C 180,E1 -26595.348,E2 -26595.348} C_VEL
LIN {X 0,Y 224.14,Z 851.365,A -85,B 0,C 180,E1 -26599.321,E2 -26599.321} C_VEL
LIN {X 0,Y 234.176,Z 838.083,A -85,B 0,C 180,E1 -26602.578,E2 -26602.578} C_VEL
LIN {X 0,Y 244.444,Z 823.012,A -85,B 0,C 180,E1 -26605.51,E2 -26605.51} C_VEL
LIN {X 0,Y 254.128,Z 807.056,A -85,B 0,C 180,E1 -26607.984,E2 -26607.984} C_VEL
LIN {X 0,Y 263.412,Z 789.596,A -85,B 0,C 180,E1 -26610.154,E2 -26610.154} C_VEL
LIN {X 0,Y 271.811,Z 771.185,A -85,B 0,C 180,E1 -26611.99,E2 -26611.99} C_VEL
LIN {X 0,Y 278.845,Z 752.848,A -85,B 0,C 180,E1 -26613.465,E2 -26613.465} C_VEL
LIN {X 0,Y 285.181,Z 732.612,A -85,B 0,C 180,E1 -26614.768,E2 -26614.768} C_VEL
LIN {X 0,Y 291.329,Z 707.3,A -85,B 0,C 180,E1 -26616.038,E2 -26616.038} C_VEL
LIN {X 0,Y 299.972,Z 668.118,A -85,B 0,C 180,E1 -26617.588,E2 -26617.588} C_VEL
LIN {X 0,Y 308.109,Z 627.632,A -85,B 0,C 180,E1 -26618.765,E2 -26618.765} C_VEL
LIN {X 0,Y 315.744,Z 582.648,A -85,B 0,C 180,E1 -26619.777,E2 -26619.777} C_VEL
LIN {X 0,Y 321.542,Z 538.915,A -85,B 0,C 180,E1 -26620.605,E2 -26620.605} C_VEL
LIN {X 0,Y 328.061,Z 477.459,A -85,B 0,C 180,E1 -26621.628,E2 -26621.628} C_VEL
LIN {X 0,Y 330.414,Z 467.626,A -85,B 0,C 180,E1 -26621.879,E2 -26621.879} C_VEL
LIN {X 0,Y 328.768,Z 458.367,A -85,B 0,C 180,E1 -26625.018,E2 -26625.018} C_VEL
LIN {X 0,Y 327.363,Z 450.758,A -85,B 0,C 180,E1 -26628.281,E2 -26628.281} C_VEL
LIN {X 0,Y 326.436,Z 444.962,A -85,B 0,C 180,E1 -26631.545,E2 -26631.545} C_VEL
LIN {X 0,Y 326.01,Z 441.627,A -85,B 0,C 180,E1 -26634.191,E2 -26634.191} C_VEL
LIN {X 0,Y 326.136,Z 438.493,A -85,B 0,C 180,E1 -26637.716,E2 -26637.716} C_VEL
LIN {X 0,Y 327.092,Z 437.825,A -85,B 0,C 180,E1 -26642.278,E2 -26642.278} C_VEL
LIN {X 0,Y 327.678,Z 438.351,A -85,B 0,C 180,E1 -26643.849,E2 -26643.849} C_VEL
LIN {X 0,Y 327.603,Z 442.751,A -85,B 0,C 180,E1 -26645.334,E2 -26645.334} C_VEL
LIN {X 0,Y 327.409,Z 447.272,A -85,B 0,C 180,E1 -26646.437,E2 -26646.437} C_VEL
LIN {X 0,Y 326.255,Z 463.463,A -85,B 0,C 180,E1 -26649.151,E2 -26649.151} C_VEL
LIN {X 0,Y 326.362,Z 466.874,A -85,B 0,C 180,E1 -26649.929,E2 -26649.929} C_VEL
LIN {X 0,Y 326.397,Z 467.982,A -85,B 0,C 180,E1 -26650.166,E2 -26650.166} C_VEL
LIN {X 0,Y 312.259,Z 540.346,A -85,B 0,C 180,E1 -26651.87,E2 -26651.87} C_VEL
LIN {X 0,Y 305.28,Z 606.43,A -85,B 0,C 180,E1 -26653.198,E2 -26653.198} C_VEL
LIN {X 0,Y 299.526,Z 644.526,A -85,B 0,C 180,E1 -26654.004,E2 -26654.004} C_VEL
LIN {X 0,Y 292.237,Z 681.798,A -85,B 0,C 180,E1 -26654.986,E2 -26654.986} C_VEL
LIN {X 0,Y 284.118,Z 715.882,A -85,B 0,C 180,E1 -26656.103,E2 -26656.103} C_VEL
LIN {X 0,Y 274.729,Z 750.047,A -85,B 0,C 180,E1 -26657.53,E2 -26657.53} C_VEL
LIN {X 0,Y 265.655,Z 779.505,A -85,B 0,C 180,E1 -26659.138,E2 -26659.138} C_VEL
LIN {X 0,Y 258.296,Z 798.949,A -85,B 0,C 180,E1 -26660.478,E2 -26660.478} C_VEL
LIN {X 0,Y 249.49,Z 818.505,A -85,B 0,C 180,E1 -26662.213,E2 -26662.213} C_VEL
LIN {X 0,Y 240.123,Z 836.275,A -85,B 0,C 180,E1 -26664.226,E2 -26664.226} C_VEL
LIN {X 0,Y 229.924,Z 853.23,A -85,B 0,C 180,E1 -26666.662,E2 -26666.662} C_VEL
LIN {X 0,Y 219.29,Z 869.139,A -85,B 0,C 180,E1 -26669.6,E2 -26669.6} C_VEL
LIN {X 0,Y 208.732,Z 883.621,A -85,B 0,C 180,E1 -26673.039,E2 -26673.039} C_VEL
LIN {X 0,Y 198.182,Z 897.046,A -85,B 0,C 180,E1 -26677.14,E2 -26677.14} C_VEL
LIN {X 0,Y 187.748,Z 909.77,A -85,B 0,C 180,E1 -26682.246,E2 -26682.246} C_VEL
LIN {X 0,Y 178.855,Z 920.4,A -85,B 0,C 180,E1 -26687.867,E2 -26687.867} C_VEL
LIN {X 0,Y 171.118,Z 930.067,A -85,B 0,C 180,E1 -26694.656,E2 -26694.656} C_VEL
LIN {X 0,Y 165.718,Z 937.68,A -85,B 0,C 180,E1 -26701.925,E2 -26701.925} C_VEL
LIN {X 0,Y 162.719,Z 943.473,A -85,B 0,C 180,E1 -26709.497,E2 -26709.497} C_VEL
LIN {X 0,Y 161.934,Z 947.595,A -85,B 0,C 180,E1 -26717.318,E2 -26717.318} C_VEL
LIN {X 0,Y 162.628,Z 949.723,A -85,B 0,C 180,E1 -26724.001,E2 -26724.001} C_VEL
LIN {X 0,Y 163.282,Z 950.365,A -85,B 0,C 180,E1 -26728.597,E2 -26728.597} C_VEL
LIN {X 0,Y 163.17,Z 950.261,A -85,B 0,C 180,E1 -26732.81,E2 -26732.81} C_VEL
LIN {X 0,Y 162.418,Z 948.979,A -85,B 0,C 180,E1 -26738.854,E2 -26738.854} C_VEL
LIN {X 0,Y 162.552,Z 945.843,A -85,B 0,C 180,E1 -26746.437,E2 -26746.437} C_VEL
LIN {X 0,Y 162.923,Z 944.984,A -85,B 0,C 180,E1 -26748.611,E2 -26748.611} C_VEL
LIN {X 0,Y 167.484,Z 943.728,A -85,B 0,C 180,E1 -26760.099,E2 -26760.099} C_VEL
LIN {X 0,Y 177.688,Z 940.769,A -85,B 0,C 180,E1 -26770.326,E2 -26770.326} C_VEL
LIN {X 0,Y 197.239,Z 935.36,A -85,B 0,C 180,E1 -26780.862,E2 -26780.862} C_VEL
LIN {X 0,Y 204.404,Z 933.345,A -85,B 0,C 180,E1 -26783.594,E2 -26783.594} C_VEL
LIN {X 0,Y 190.818,Z 930.638,A -85,B 0,C 180,E1 -26789.101,E2 -26789.101} C_VEL
LIN {X 0,Y 179.821,Z 926.238,A -85,B 0,C 180,E1 -26795.352,E2 -26795.352} C_VEL
LIN {X 0,Y 171.811,Z 920.292,A -85,B 0,C 180,E1 -26802.034,E2 -26802.034} C_VEL
LIN {X 0,Y 166.376,Z 912.489,A -85,B 0,C 180,E1 -26809.263,E2 -26809.263} C_VEL
LIN {X 0,Y 163.582,Z 903.556,A -85,B 0,C 180,E1 -26816.145,E2 -26816.145} C_VEL
LIN {X 0,Y 162.558,Z 893.783,A -85,B 0,C 180,E1 -26822.468,E2 -26822.468} C_VEL
LIN {X 0,Y 162.772,Z 881.994,A -85,B 0,C 180,E1 -26828.834,E2 -26828.834} C_VEL
LIN {X 0,Y 163.456,Z 874.182,A -85,B 0,C 180,E1 -26832.542,E2 -26832.542} C_VEL
LIN {X 0,Y 164.692,Z 873.5,A -85,B 0,C 180,E1 -26834.773,E2 -26834.773} C_VEL
LIN {X 0,Y 166.338,Z 872.586,A -85,B 0,C 180,E1 -26836.411,E2 -26836.411} C_VEL
LIN {X 0,Y 168.481,Z 871.593,A -85,B 0,C 180,E1 -26838.692,E2 -26838.692} C_VEL
LIN {X 0,Y 169.996,Z 870.896,A -85,B 0,C 180,E1 -26839.947,E2 -26839.947} C_VEL
LIN {X 0,Y 173.185,Z 869.561,A -85,B 0,C 180,E1 -26842.399,E2 -26842.399} C_VEL
LIN {X 0,Y 178.171,Z 867.644,A -85,B 0,C 180,E1 -26845.603,E2 -26845.603} C_VEL
LIN {X 0,Y 183.824,Z 865.611,A -85,B 0,C 180,E1 -26848.599,E2 -26848.599} C_VEL
LIN {X 0,Y 196.302,Z 861.336,A -85,B 0,C 180,E1 -26853.725,E2 -26853.725} C_VEL
LIN {X 0,Y 213.962,Z 855.173,A -85,B 0,C 180,E1 -26858.771,E2 -26858.771} C_VEL
LIN {X 0,Y 217.717,Z 853.818,A -85,B 0,C 180,E1 -26859.619,E2 -26859.619} C_VEL
LIN {X 0,Y 206.463,Z 866.757,A -85,B 0,C 180,E1 -26863.832,E2 -26863.832} C_VEL
LIN {X 0,Y 195.999,Z 877.812,A -85,B 0,C 180,E1 -26868.584,E2 -26868.584} C_VEL
LIN {X 0,Y 186.64,Z 887.075,A -85,B 0,C 180,E1 -26873.892,E2 -26873.892} C_VEL
LIN {X 0,Y 178.646,Z 894.647,A -85,B 0,C 180,E1 -26879.752,E2 -26879.752} C_VEL
LIN {X 0,Y 172.072,Z 900.773,A -85,B 0,C 180,E1 -26886.362,E2 -26886.362} C_VEL
LIN {X 0,Y 167.41,Z 905.164,A -85,B 0,C 180,E1 -26893.34,E2 -26893.34} C_VEL
LIN {X 0,Y 164.64,Z 907.919,A -85,B 0,C 180,E1 -26900.562,E2 -26900.562} C_VEL
LIN {X 0,Y 163.516,Z 909.125,A -85,B 0,C 180,E1 -26907.897,E2 -26907.897} C_VEL
LIN {X 0,Y 163.758,Z 908.882,A -85,B 0,C 180,E1 -26914.904,E2 -26914.904} C_VEL
LIN {X 0,Y 165.345,Z 907.279,A -85,B 0,C 180,E1 -26921.865,E2 -26921.865} C_VEL
LIN {X 0,Y 168.914,Z 903.828,A -85,B 0,C 180,E1 -26929.359,E2 -26929.359} C_VEL
LIN {X 0,Y 174.289,Z 898.843,A -85,B 0,C 180,E1 -26936.215,E2 -26936.215} C_VEL
LIN {X 0,Y 181.575,Z 892.061,A -85,B 0,C 180,E1 -26942.66,E2 -26942.66} C_VEL
LIN {X 0,Y 190.656,Z 883.332,A -85,B 0,C 180,E1 -26948.615,E2 -26948.615} C_VEL
LIN {X 0,Y 200.81,Z 873.018,A -85,B 0,C 180,E1 -26953.798,E2 -26953.798} C_VEL
LIN {X 0,Y 211.3,Z 861.561,A -85,B 0,C 180,E1 -26958.146,E2 -26958.146} C_VEL
LIN {X 0,Y 222.217,Z 848.54,A -85,B 0,C 180,E1 -26961.946,E2 -26961.946} C_VEL
LIN {X 0,Y 232.801,Z 834.608,A -85,B 0,C 180,E1 -26965.12,E2 -26965.12} C_VEL
LIN {X 0,Y 243.208,Z 819.289,A -85,B 0,C 180,E1 -26967.878,E2 -26967.878} C_VEL
LIN {X 0,Y 252.927,Z 803.13,A -85,B 0,C 180,E1 -26970.197,E2 -26970.197} C_VEL
LIN {X 0,Y 261.796,Z 786.253,A -85,B 0,C 180,E1 -26972.151,E2 -26972.151} C_VEL
LIN {X 0,Y 270.198,Z 767.496,A -85,B 0,C 180,E1 -26973.898,E2 -26973.898} C_VEL
LIN {X 0,Y 277.309,Z 748.444,A -85,B 0,C 180,E1 -26975.317,E2 -26975.317} C_VEL
LIN {X 0,Y 283.179,Z 728.923,A -85,B 0,C 180,E1 -26976.484,E2 -26976.484} C_VEL
LIN {X 0,Y 292.148,Z 691.357,A -85,B 0,C 180,E1 -26978.198,E2 -26978.198} C_VEL
LIN {X 0,Y 300.79,Z 651.633,A -85,B 0,C 180,E1 -26979.555,E2 -26979.555} C_VEL
LIN {X 0,Y 309.071,Z 608.575,A -85,B 0,C 180,E1 -26980.621,E2 -26980.621} C_VEL
LIN {X 0,Y 315.944,Z 564.301,A -85,B 0,C 180,E1 -26981.521,E2 -26981.521} C_VEL
LIN {X 0,Y 321.34,Z 518.138,A -85,B 0,C 180,E1 -26982.315,E2 -26982.315} C_VEL
LIN {X 0,Y 325.459,Z 480.137,A -85,B 0,C 180,E1 -26982.93,E2 -26982.93} C_VEL
LIN {X 0,Y 327.356,Z 472.231,A -85,B 0,C 180,E1 -26983.132,E2 -26983.132} C_VEL
LIN {X 0,Y 326.031,Z 463.911,A -85,B 0,C 180,E1 -26986.114,E2 -26986.114} C_VEL
LIN {X 0,Y 324.966,Z 457.487,A -85,B 0,C 180,E1 -26989.002,E2 -26989.002} C_VEL
LIN {X 0,Y 324.283,Z 452.166,A -85,B 0,C 180,E1 -26992.113,E2 -26992.113} C_VEL
LIN {X 0,Y 324.015,Z 449.197,A -85,B 0,C 180,E1 -26994.51,E2 -26994.51} C_VEL
LIN {X 0,Y 324.198,Z 446.224,A -85,B 0,C 180,E1 -26997.879,E2 -26997.879} C_VEL
LIN {X 0,Y 325.29,Z 445.62,A -85,B 0,C 180,E1 -27002.29,E2 -27002.29} C_VEL
LIN {X 0,Y 325.711,Z 446.095,A -85,B 0,C 180,E1 -27003.52,E2 -27003.52} C_VEL
LIN {X 0,Y 325.714,Z 457.481,A -85,B 0,C 180,E1 -27007.231,E2 -27007.231} C_VEL
LIN {X 0,Y 326.362,Z 466.874,A -85,B 0,C 180,E1 -27009.929,E2 -27009.929} C_VEL
LIN {X 0,Y 326.236,Z 469.482,A -85,B 0,C 180,E1 -27010.306,E2 -27010.306} C_VEL
LIN {X 0,Y 325.497,Z 473.821,A -85,B 0,C 180,E1 -27010.482,E2 -27010.482} C_VEL
LIN {X 0,Y 323.928,Z 480.199,A -85,B 0,C 180,E1 -27010.355,E2 -27010.355} C_VEL
LIN {X 0,Y 319.801,Z 494.115,A -85,B 0,C 180,E1 -27009.598,E2 -27009.598} C_VEL
LIN {X 0,Y 318.284,Z 500.243,A -85,B 0,C 180,E1 -27009.5,E2 -27009.5} C_VEL
LIN {X 0,Y 318.03,Z 501.48,A -85,B 0,C 180,E1 -27009.52,E2 -27009.52} C_VEL
LIN {X 0,Y 310.898,Z 537.494,A -85,B 0,C 180,E1 -27010.367,E2 -27010.367} C_VEL
LIN {X 0,Y 303.693,Z 603.933,A -85,B 0,C 180,E1 -27011.68,E2 -27011.68} C_VEL
LIN {X 0,Y 297.888,Z 641.792,A -85,B 0,C 180,E1 -27012.458,E2 -27012.458} C_VEL
LIN {X 0,Y 290.39,Z 679.604,A -85,B 0,C 180,E1 -27013.413,E2 -27013.413} C_VEL
LIN {X 0,Y 281.841,Z 714.965,A -85,B 0,C 180,E1 -27014.525,E2 -27014.525} C_VEL
LIN {X 0,Y 272.159,Z 749.508,A -85,B 0,C 180,E1 -27015.92,E2 -27015.92} C_VEL
LIN {X 0,Y 262.796,Z 779.154,A -85,B 0,C 180,E1 -27017.493,E2 -27017.493} C_VEL
LIN {X 0,Y 255.108,Z 798.754,A -85,B 0,C 180,E1 -27018.817,E2 -27018.817} C_VEL
LIN {X 0,Y 246.068,Z 818.016,A -85,B 0,C 180,E1 -27020.507,E2 -27020.507} C_VEL
LIN {X 0,Y 236.339,Z 835.816,A -85,B 0,C 180,E1 -27022.488,E2 -27022.488} C_VEL
LIN {X 0,Y 225.529,Z 853.14,A -85,B 0,C 180,E1 -27024.952,E2 -27024.952} C_VEL
LIN {X 0,Y 213.681,Z 870.088,A -85,B 0,C 180,E1 -27028.108,E2 -27028.108} C_VEL
LIN {X 0,Y 202.24,Z 884.969,A -85,B 0,C 180,E1 -27031.747,E2 -27031.747} C_VEL
LIN {X 0,Y 190.763,Z 898.788,A -85,B 0,C 180,E1 -27036.177,E2 -27036.177} C_VEL
LIN {X 0,Y 180.044,Z 911.037,A -85,B 0,C 180,E1 -27041.433,E2 -27041.433} C_VEL
LIN {X 0,Y 170.49,Z 921.75,A -85,B 0,C 180,E1 -27047.589,E2 -27047.589} C_VEL
LIN {X 0,Y 162.49,Z 931.148,A -85,B 0,C 180,E1 -27054.928,E2 -27054.928} C_VEL
LIN {X 0,Y 157.152,Z 938.44,A -85,B 0,C 180,E1 -27062.735,E2 -27062.735} C_VEL
LIN {X 0,Y 154.396,Z 943.938,A -85,B 0,C 180,E1 -27071,E2 -27071} C_VEL
LIN {X 0,Y 154.042,Z 947.377,A -85,B 0,C 180,E1 -27078.771,E2 -27078.771} C_VEL
LIN {X 0,Y 154.925,Z 949.061,A -85,B 0,C 180,E1 -27085.558,E2 -27085.558} C_VEL
LIN {X 0,Y 155.419,Z 949.442,A -85,B 0,C 180,E1 -27090,E2 -27090} C_VEL
LIN {X 0,Y 154.951,Z 948.992,A -85,B 0,C 180,E1 -27094.812,E2 -27094.812} C_VEL
LIN {X 0,Y 154.303,Z 947.253,A -85,B 0,C 180,E1 -27101.589,E2 -27101.589} C_VEL
LIN {X 0,Y 155.177,Z 943.6,A -85,B 0,C 180,E1 -27109.577,E2 -27109.577} C_VEL
LIN {X 0,Y 155.685,Z 942.909,A -85,B 0,C 180,E1 -27111.367,E2 -27111.367} C_VEL
LIN {X 0,Y 162.106,Z 941.586,A -85,B 0,C 180,E1 -27123.72,E2 -27123.72} C_VEL
LIN {X 0,Y 175.717,Z 938.278,A -85,B 0,C 180,E1 -27134.879,E2 -27134.879} C_VEL
LIN {X 0,Y 194.155,Z 933.809,A -85,B 0,C 180,E1 -27143.621,E2 -27143.621} C_VEL
LIN {X 0,Y 180.797,Z 930.272,A -85,B 0,C 180,E1 -27149.416,E2 -27149.416} C_VEL
LIN {X 0,Y 170.046,Z 924.983,A -85,B 0,C 180,E1 -27156.063,E2 -27156.063} C_VEL
LIN {X 0,Y 162.406,Z 918.195,A -85,B 0,C 180,E1 -27163.18,E2 -27163.18} C_VEL
LIN {X 0,Y 157.612,Z 909.934,A -85,B 0,C 180,E1 -27170.506,E2 -27170.506} C_VEL
LIN {X 0,Y 155.194,Z 900.202,A -85,B 0,C 180,E1 -27177.785,E2 -27177.785} C_VEL
LIN {X 0,Y 154.524,Z 889.524,A -85,B 0,C 180,E1 -27184.454,E2 -27184.454} C_VEL
LIN {X 0,Y 154.874,Z 880.228,A -85,B 0,C 180,E1 -27189.476,E2 -27189.476} C_VEL
LIN {X 0,Y 155.771,Z 879.544,A -85,B 0,C 180,E1 -27191.853,E2 -27191.853} C_VEL
LIN {X 0,Y 157.17,Z 878.655,A -85,B 0,C 180,E1 -27193.615,E2 -27193.615} C_VEL
LIN {X 0,Y 159.294,Z 877.528,A -85,B 0,C 180,E1 -27196.408,E2 -27196.408} C_VEL
LIN {X 0,Y 163.019,Z 875.829,A -85,B 0,C 180,E1 -27200.089,E2 -27200.089} C_VEL
LIN {X 0,Y 167.509,Z 874.038,A -85,B 0,C 180,E1 -27203.574,E2 -27203.574} C_VEL
LIN {X 0,Y 177.965,Z 870.352,A -85,B 0,C 180,E1 -27209.632,E2 -27209.632} C_VEL
LIN {X 0,Y 192.867,Z 865.444,A -85,B 0,C 180,E1 -27215.496,E2 -27215.496} C_VEL
LIN {X 0,Y 207.636,Z 860.681,A -85,B 0,C 180,E1 -27219.709,E2 -27219.709} C_VEL
LIN {X 0,Y 196.368,Z 872.639,A -85,B 0,C 180,E1 -27224.113,E2 -27224.113} C_VEL
LIN {X 0,Y 185.576,Z 883.186,A -85,B 0,C 180,E1 -27229.311,E2 -27229.311} C_VEL
LIN {X 0,Y 175.811,Z 892.134,A -85,B 0,C 180,E1 -27235.338,E2 -27235.338} C_VEL
LIN {X 0,Y 167.874,Z 899.118,A -85,B 0,C 180,E1 -27241.93,E2 -27241.93} C_VEL
LIN {X 0,Y 161.913,Z 904.303,A -85,B 0,C 180,E1 -27249.011,E2 -27249.011} C_VEL
LIN {X 0,Y 157.98,Z 907.815,A -85,B 0,C 180,E1 -27256.456,E2 -27256.456} C_VEL
LIN {X 0,Y 155.961,Z 909.742,A -85,B 0,C 180,E1 -27264.112,E2 -27264.112} C_VEL
LIN {X 0,Y 155.547,Z 910.174,A -85,B 0,C 180,E1 -27271.473,E2 -27271.473} C_VEL
LIN {X 0,Y 156.513,Z 909.256,A -85,B 0,C 180,E1 -27278.819,E2 -27278.819} C_VEL
LIN {X 0,Y 159.212,Z 906.786,A -85,B 0,C 180,E1 -27286.416,E2 -27286.416} C_VEL
LIN {X 0,Y 164.178,Z 902.442,A -85,B 0,C 180,E1 -27294.082,E2 -27294.082} C_VEL
LIN {X 0,Y 170.972,Z 896.543,A -85,B 0,C 180,E1 -27300.974,E2 -27300.974} C_VEL
LIN {X 0,Y 179.703,Z 888.775,A -85,B 0,C 180,E1 -27307.336,E2 -27307.336} C_VEL
LIN {X 0,Y 189.691,Z 879.429,A -85,B 0,C 180,E1 -27312.887,E2 -27312.887} C_VEL
LIN {X 0,Y 200.352,Z 868.737,A -85,B 0,C 180,E1 -27317.614,E2 -27317.614} C_VEL
LIN {X 0,Y 211.504,Z 856.553,A -85,B 0,C 180,E1 -27321.699,E2 -27321.699} C_VEL
LIN {X 0,Y 222.123,Z 843.831,A -85,B 0,C 180,E1 -27325.012,E2 -27325.012} C_VEL
LIN {X 0,Y 233.302,Z 828.879,A -85,B 0,C 180,E1 -27328.059,E2 -27328.059} C_VEL
LIN {X 0,Y 243.856,Z 812.959,A -85,B 0,C 180,E1 -27330.612,E2 -27330.612} C_VEL
LIN {X 0,Y 253.878,Z 795.636,A -85,B 0,C 180,E1 -27332.815,E2 -27332.815} C_VEL
LIN {X 0,Y 262.798,Z 777.688,A -85,B 0,C 180,E1 -27334.64,E2 -27334.64} C_VEL
LIN {X 0,Y 270.565,Z 759.168,A -85,B 0,C 180,E1 -27336.156,E2 -27336.156} C_VEL
LIN {X 0,Y 277.219,Z 739.86,A -85,B 0,C 180,E1 -27337.422,E2 -27337.422} C_VEL
LIN {X 0,Y 282.976,Z 718.593,A -85,B 0,C 180,E1 -27338.533,E2 -27338.533} C_VEL
LIN {X 0,Y 291.879,Z 681.09,A -85,B 0,C 180,E1 -27340.075,E2 -27340.075} C_VEL
LIN {X 0,Y 300.204,Z 642.664,A -85,B 0,C 180,E1 -27341.255,E2 -27341.255} C_VEL
LIN {X 0,Y 308.37,Z 599.066,A -85,B 0,C 180,E1 -27342.248,E2 -27342.248} C_VEL
LIN {X 0,Y 314.798,Z 555.878,A -85,B 0,C 180,E1 -27343.069,E2 -27343.069} C_VEL
LIN {X 0,Y 322.131,Z 488.972,A -85,B 0,C 180,E1 -27344.146,E2 -27344.146} C_VEL
LIN {X 0,Y 323.313,Z 481.69,A -85,B 0,C 180,E1 -27344.277,E2 -27344.277} C_VEL
LIN {X 0,Y 324.454,Z 476.957,A -85,B 0,C 180,E1 -27344.402,E2 -27344.402} C_VEL
LIN {X 0,Y 323.375,Z 469.3,A -85,B 0,C 180,E1 -27347.318,E2 -27347.318} C_VEL
LIN {X 0,Y 322.503,Z 462.664,A -85,B 0,C 180,E1 -27350.542,E2 -27350.542} C_VEL
LIN {X 0,Y 322.062,Z 458.355,A -85,B 0,C 180,E1 -27353.457,E2 -27353.457} C_VEL
LIN {X 0,Y 322.023,Z 456.468,A -85,B 0,C 180,E1 -27355.191,E2 -27355.191} C_VEL
LIN {X 0,Y 322.392,Z 453.985,A -85,B 0,C 180,E1 -27358.045,E2 -27358.045} C_VEL
LIN {X 0,Y 323.478,Z 453.423,A -85,B 0,C 180,E1 -27362.48,E2 -27362.48} C_VEL
LIN {X 0,Y 323.726,Z 453.75,A -85,B 0,C 180,E1 -27363.143,E2 -27363.143} C_VEL
LIN {X 0,Y 323.619,Z 464.22,A -85,B 0,C 180,E1 -27366.564,E2 -27366.564} C_VEL
LIN {X 0,Y 323.99,Z 472.347,A -85,B 0,C 180,E1 -27368.874,E2 -27368.874} C_VEL
LIN {X 0,Y 318.03,Z 501.48,A -85,B 0,C 180,E1 -27369.52,E2 -27369.52} C_VEL
LIN {X 0,Y 316.548,Z 507.968,A -85,B 0,C 180,E1 -27369.518,E2 -27369.518} C_VEL
LIN {X 0,Y 311.017,Z 528.159,A -85,B 0,C 180,E1 -27368.841,E2 -27368.841} C_VEL
LIN {X 0,Y 309.629,Z 535.804,A -85,B 0,C 180,E1 -27368.874,E2 -27368.874} C_VEL
LIN {X 0,Y 302.321,Z 601.428,A -85,B 0,C 180,E1 -27370.147,E2 -27370.147} C_VEL
LIN {X 0,Y 296.532,Z 638.71,A -85,B 0,C 180,E1 -27370.889,E2 -27370.889} C_VEL
LIN {X 0,Y 289.033,Z 676.098,A -85,B 0,C 180,E1 -27371.788,E2 -27371.788} C_VEL
LIN {X 0,Y 280.532,Z 711.081,A -85,B 0,C 180,E1 -27372.826,E2 -27372.826} C_VEL
LIN {X 0,Y 270.691,Z 746.056,A -85,B 0,C 180,E1 -27374.156,E2 -27374.156} C_VEL
LIN {X 0,Y 261.149,Z 775.901,A -85,B 0,C 180,E1 -27375.646,E2 -27375.646} C_VEL
LIN {X 0,Y 253.42,Z 795.529,A -85,B 0,C 180,E1 -27376.902,E2 -27376.902} C_VEL
LIN {X 0,Y 244.549,Z 814.389,A -85,B 0,C 180,E1 -27378.454,E2 -27378.454} C_VEL
LIN {X 0,Y 234.584,Z 832.421,A -85,B 0,C 180,E1 -27380.327,E2 -27380.327} C_VEL
LIN {X 0,Y 223.313,Z 850.179,A -85,B 0,C 180,E1 -27382.725,E2 -27382.725} C_VEL
LIN {X 0,Y 211.744,Z 866.408,A -85,B 0,C 180,E1 -27385.587,E2 -27385.587} C_VEL
LIN {X 0,Y 199.981,Z 881.31,A -85,B 0,C 180,E1 -27389.012,E2 -27389.012} C_VEL
LIN {X 0,Y 187.826,Z 895.418,A -85,B 0,C 180,E1 -27393.302,E2 -27393.302} C_VEL
LIN {X 0,Y 176.834,Z 907.448,A -85,B 0,C 180,E1 -27398.191,E2 -27398.191} C_VEL
LIN {X 0,Y 166.405,Z 918.484,A -85,B 0,C 180,E1 -27404.188,E2 -27404.188} C_VEL
LIN {X 0,Y 157.691,Z 927.835,A -85,B 0,C 180,E1 -27411.117,E2 -27411.117} C_VEL
LIN {X 0,Y 151.147,Z 935.497,A -85,B 0,C 180,E1 -27418.936,E2 -27418.936} C_VEL
LIN {X 0,Y 147.215,Z 941.475,A -85,B 0,C 180,E1 -27427.476,E2 -27427.476} C_VEL
LIN {X 0,Y 145.987,Z 945.594,A -85,B 0,C 180,E1 -27436.13,E2 -27436.13} C_VEL
LIN {X 0,Y 146.665,Z 947.759,A -85,B 0,C 180,E1 -27443.738,E2 -27443.738} C_VEL
LIN {X 0,Y 147.416,Z 948.383,A -85,B 0,C 180,E1 -27448.834,E2 -27448.834} C_VEL
LIN {X 0,Y 147.236,Z 948.249,A -85,B 0,C 180,E1 -27453.115,E2 -27453.115} C_VEL
LIN {X 0,Y 146.413,Z 946.928,A -85,B 0,C 180,E1 -27459.831,E2 -27459.831} C_VEL
LIN {X 0,Y 146.896,Z 943.753,A -85,B 0,C 180,E1 -27468.247,E2 -27468.247} C_VEL
LIN {X 0,Y 148.736,Z 940.738,A -85,B 0,C 180,E1 -27474.21,E2 -27474.21} C_VEL
LIN {X 0,Y 155.377,Z 939.69,A -85,B 0,C 180,E1 -27485.393,E2 -27485.393} C_VEL
LIN {X 0,Y 171.57,Z 936.487,A -85,B 0,C 180,E1 -27497.744,E2 -27497.744} C_VEL
LIN {X 0,Y 184.071,Z 933.865,A -85,B 0,C 180,E1 -27503.588,E2 -27503.588} C_VEL
LIN {X 0,Y 170.784,Z 929.414,A -85,B 0,C 180,E1 -27509.768,E2 -27509.768} C_VEL
LIN {X 0,Y 160.311,Z 923.283,A -85,B 0,C 180,E1 -27516.862,E2 -27516.862} C_VEL
LIN {X 0,Y 152.813,Z 915.245,A -85,B 0,C 180,E1 -27524.827,E2 -27524.827} C_VEL
LIN {X 0,Y 148.626,Z 905.995,A -85,B 0,C 180,E1 -27532.656,E2 -27532.656} C_VEL
LIN {X 0,Y 146.843,Z 895.8,A -85,B 0,C 180,E1 -27540,E2 -27540} C_VEL
LIN {X 0,Y 146.572,Z 886.134,A -85,B 0,C 180,E1 -27546.07,E2 -27546.07} C_VEL
LIN {X 0,Y 147.399,Z 885.194,A -85,B 0,C 180,E1 -27548.976,E2 -27548.976} C_VEL
LIN {X 0,Y 148.317,Z 884.486,A -85,B 0,C 180,E1 -27550.488,E2 -27550.488} C_VEL
LIN {X 0,Y 149.995,Z 883.391,A -85,B 0,C 180,E1 -27553.492,E2 -27553.492} C_VEL
LIN {X 0,Y 153.551,Z 881.562,A -85,B 0,C 180,E1 -27557.822,E2 -27557.822} C_VEL
LIN {X 0,Y 157.086,Z 880.085,A -85,B 0,C 180,E1 -27561.274,E2 -27561.274} C_VEL
LIN {X 0,Y 167.216,Z 876.434,A -85,B 0,C 180,E1 -27568.19,E2 -27568.19} C_VEL
LIN {X 0,Y 180.712,Z 872.139,A -85,B 0,C 180,E1 -27574.359,E2 -27574.359} C_VEL
LIN {X 0,Y 196.903,Z 867.132,A -85,B 0,C 180,E1 -27579.478,E2 -27579.478} C_VEL
LIN {X 0,Y 197.669,Z 866.971,A -85,B 0,C 180,E1 -27579.746,E2 -27579.746} C_VEL
LIN {X 0,Y 186.217,Z 878.185,A -85,B 0,C 180,E1 -27584.427,E2 -27584.427} C_VEL
LIN {X 0,Y 175.474,Z 887.891,A -85,B 0,C 180,E1 -27589.916,E2 -27589.916} C_VEL
LIN {X 0,Y 165.864,Z 896.049,A -85,B 0,C 180,E1 -27596.316,E2 -27596.316} C_VEL
LIN {X 0,Y 157.881,Z 902.574,A -85,B 0,C 180,E1 -27603.684,E2 -27603.684} C_VEL
LIN {X 0,Y 152.208,Z 907.194,A -85,B 0,C 180,E1 -27611.619,E2 -27611.619} C_VEL
LIN {X 0,Y 148.973,Z 909.931,A -85,B 0,C 180,E1 -27619.559,E2 -27619.559} C_VEL
LIN {X 0,Y 147.652,Z 911.127,A -85,B 0,C 180,E1 -27627.671,E2 -27627.671} C_VEL
LIN {X 0,Y 147.938,Z 910.887,A -85,B 0,C 180,E1 -27635.429,E2 -27635.429} C_VEL
LIN {X 0,Y 149.799,Z 909.291,A -85,B 0,C 180,E1 -27643.117,E2 -27643.117} C_VEL
LIN {X 0,Y 153.953,Z 905.858,A -85,B 0,C 180,E1 -27651.328,E2 -27651.328} C_VEL
LIN {X 0,Y 160.113,Z 900.891,A -85,B 0,C 180,E1 -27658.741,E2 -27658.741} C_VEL
LIN {X 0,Y 168.341,Z 894.131,A -85,B 0,C 180,E1 -27665.597,E2 -27665.597} C_VEL
LIN {X 0,Y 177.935,Z 885.906,A -85,B 0,C 180,E1 -27671.536,E2 -27671.536} C_VEL
LIN {X 0,Y 188.44,Z 876.302,A -85,B 0,C 180,E1 -27676.631,E2 -27676.631} C_VEL
LIN {X 0,Y 200.111,Z 864.677,A -85,B 0,C 180,E1 -27681.213,E2 -27681.213} C_VEL
LIN {X 0,Y 212.085,Z 851.535,A -85,B 0,C 180,E1 -27685.118,E2 -27685.118} C_VEL
LIN {X 0,Y 223.366,Z 837.762,A -85,B 0,C 180,E1 -27688.269,E2 -27688.269} C_VEL
LIN {X 0,Y 234.763,Z 822.076,A -85,B 0,C 180,E1 -27691.068,E2 -27691.068} C_VEL
LIN {X 0,Y 245.041,Z 806,A -85,B 0,C 180,E1 -27693.333,E2 -27693.333} C_VEL
LIN {X 0,Y 254.379,Z 789.217,A -85,B 0,C 180,E1 -27695.229,E2 -27695.229} C_VEL
LIN {X 0,Y 262.679,Z 771.838,A -85,B 0,C 180,E1 -27696.82,E2 -27696.82} C_VEL
LIN {X 0,Y 270.267,Z 752.827,A -85,B 0,C 180,E1 -27698.219,E2 -27698.219} C_VEL
LIN {X 0,Y 276.477,Z 733.625,A -85,B 0,C 180,E1 -27699.354,E2 -27699.354} C_VEL
LIN {X 0,Y 285.763,Z 697.265,A -85,B 0,C 180,E1 -27701,E2 -27701} C_VEL
LIN {X 0,Y 294.593,Z 658.964,A -85,B 0,C 180,E1 -27702.299,E2 -27702.299} C_VEL
LIN {X 0,Y 302.737,Z 618.996,A -85,B 0,C 180,E1 -27703.279,E2 -27703.279} C_VEL
LIN {X 0,Y 309.889,Z 576.444,A -85,B 0,C 180,E1 -27704.123,E2 -27704.123} C_VEL
LIN {X 0,Y 315.402,Z 533.551,A -85,B 0,C 180,E1 -27704.846,E2 -27704.846} C_VEL
LIN {X 0,Y 320.745,Z 485.656,A -85,B 0,C 180,E1 -27705.591,E2 -27705.591} C_VEL
LIN {X 0,Y 321.688,Z 481.786,A -85,B 0,C 180,E1 -27705.693,E2 -27705.693} C_VEL
LIN {X 0,Y 320.793,Z 474.307,A -85,B 0,C 180,E1 -27708.766,E2 -27708.766} C_VEL
LIN {X 0,Y 320.211,Z 468.481,A -85,B 0,C 180,E1 -27711.922,E2 -27711.922} C_VEL
LIN {X 0,Y 320.057,Z 464.479,A -85,B 0,C 180,E1 -27714.982,E2 -27714.982} C_VEL
LIN {X 0,Y 320.519,Z 461.73,A -85,B 0,C 180,E1 -27718.212,E2 -27718.212} C_VEL
LIN {X 0,Y 321.663,Z 461.217,A -85,B 0,C 180,E1 -27722.494,E2 -27722.494} C_VEL
LIN {X 0,Y 321.72,Z 461.658,A -85,B 0,C 180,E1 -27722.85,E2 -27722.85} C_VEL
LIN {X 0,Y 321.499,Z 471.093,A -85,B 0,C 180,E1 -27725.936,E2 -27725.936} C_VEL
LIN {X 0,Y 321.594,Z 476.923,A -85,B 0,C 180,E1 -27727.57,E2 -27727.57} C_VEL
LIN {X 0,Y 309.776,Z 534.416,A -85,B 0,C 180,E1 -27728.846,E2 -27728.846} C_VEL
LIN {X 0,Y 309.629,Z 535.804,A -85,B 0,C 180,E1 -27728.874,E2 -27728.874} C_VEL
LIN {X 0,Y 308.647,Z 543.505,A -85,B 0,C 180,E1 -27728.845,E2 -27728.845} C_VEL
LIN {X 0,Y 305.43,Z 564.115,A -85,B 0,C 180,E1 -27728.078,E2 -27728.078} C_VEL
LIN {X 0,Y 304.602,Z 570.726,A -85,B 0,C 180,E1 -27728.063,E2 -27728.063} C_VEL
LIN {X 0,Y 299.515,Z 610.459,A -85,B 0,C 180,E1 -27728.828,E2 -27728.828} C_VEL
LIN {X 0,Y 293.011,Z 648.006,A -85,B 0,C 180,E1 -27729.57,E2 -27729.57} C_VEL
LIN {X 0,Y 284.888,Z 685.595,A -85,B 0,C 180,E1 -27730.491,E2 -27730.491} C_VEL
LIN {X 0,Y 276.271,Z 719.212,A -85,B 0,C 180,E1 -27731.505,E2 -27731.505} C_VEL
LIN {X 0,Y 266.563,Z 752.045,A -85,B 0,C 180,E1 -27732.769,E2 -27732.769} C_VEL
LIN {X 0,Y 258.109,Z 777.266,A -85,B 0,C 180,E1 -27734.037,E2 -27734.037} C_VEL
LIN {X 0,Y 249.689,Z 797.475,A -85,B 0,C 180,E1 -27735.325,E2 -27735.325} C_VEL
LIN {X 0,Y 240.334,Z 816.295,A -85,B 0,C 180,E1 -27736.884,E2 -27736.884} C_VEL
LIN {X 0,Y 229.783,Z 834.418,A -85,B 0,C 180,E1 -27738.784,E2 -27738.784} C_VEL
LIN {X 0,Y 218.185,Z 851.818,A -85,B 0,C 180,E1 -27741.158,E2 -27741.158} C_VEL
LIN {X 0,Y 206.701,Z 867.164,A -85,B 0,C 180,E1 -27743.899,E2 -27743.899} C_VEL
LIN {X 0,Y 195.127,Z 881.149,A -85,B 0,C 180,E1 -27747.133,E2 -27747.133} C_VEL
LIN {X 0,Y 182.758,Z 894.872,A -85,B 0,C 180,E1 -27751.316,E2 -27751.316} C_VEL
LIN {X 0,Y 170.534,Z 907.555,A -85,B 0,C 180,E1 -27756.557,E2 -27756.557} C_VEL
LIN {X 0,Y 159.443,Z 918.511,A -85,B 0,C 180,E1 -27762.801,E2 -27762.801} C_VEL
LIN {X 0,Y 150.43,Z 927.504,A -85,B 0,C 180,E1 -27769.853,E2 -27769.853} C_VEL
LIN {X 0,Y 143.494,Z 935.031,A -85,B 0,C 180,E1 -27778.023,E2 -27778.023} C_VEL
LIN {X 0,Y 139.264,Z 940.973,A -85,B 0,C 180,E1 -27787.188,E2 -27787.188} C_VEL
LIN {X 0,Y 138.021,Z 944.864,A -85,B 0,C 180,E1 -27796.169,E2 -27796.169} C_VEL
LIN {X 0,Y 138.775,Z 946.888,A -85,B 0,C 180,E1 -27804.211,E2 -27804.211} C_VEL
LIN {X 0,Y 139.501,Z 947.405,A -85,B 0,C 180,E1 -27809.179,E2 -27809.179} C_VEL
LIN {X 0,Y 139.209,Z 947.209,A -85,B 0,C 180,E1 -27813.707,E2 -27813.707} C_VEL
LIN {X 0,Y 138.396,Z 945.673,A -85,B 0,C 180,E1 -27821.249,E2 -27821.249} C_VEL
LIN {X 0,Y 139.297,Z 942.315,A -85,B 0,C 180,E1 -27830.155,E2 -27830.155} C_VEL
LIN {X 0,Y 142.085,Z 938.515,A -85,B 0,C 180,E1 -27837.221,E2 -27837.221} C_VEL
LIN {X 0,Y 151.455,Z 937.285,A -85,B 0,C 180,E1 -27849.821,E2 -27849.821} C_VEL
LIN {X 0,Y 167.908,Z 934.507,A -85,B 0,C 180,E1 -27860.728,E2 -27860.728} C_VEL
LIN {X 0,Y 173.977,Z 933.459,A -85,B 0,C 180,E1 -27863.559,E2 -27863.559} C_VEL
LIN {X 0,Y 160.793,Z 928.115,A -85,B 0,C 180,E1 -27870.167,E2 -27870.167} C_VEL
LIN {X 0,Y 150.628,Z 921.136,A -85,B 0,C 180,E1 -27877.767,E2 -27877.767} C_VEL
LIN {X 0,Y 143.831,Z 912.629,A -85,B 0,C 180,E1 -27885.918,E2 -27885.918} C_VEL
LIN {X 0,Y 140.181,Z 903.096,A -85,B 0,C 180,E1 -27893.858,E2 -27893.858} C_VEL
LIN {X 0,Y 138.747,Z 892.688,A -85,B 0,C 180,E1 -27901.239,E2 -27901.239} C_VEL
LIN {X 0,Y 138.652,Z 891.909,A -85,B 0,C 180,E1 -27902.066,E2 -27902.066} C_VEL
LIN {X 0,Y 139.357,Z 890.625,A -85,B 0,C 180,E1 -27905.765,E2 -27905.765} C_VEL
LIN {X 0,Y 139.949,Z 889.94,A -85,B 0,C 180,E1 -27907.802,E2 -27907.802} C_VEL
LIN {X 0,Y 141.861,Z 888.452,A -85,B 0,C 180,E1 -27911.795,E2 -27911.795} C_VEL
LIN {X 0,Y 151.117,Z 884.139,A -85,B 0,C 180,E1 -27922.567,E2 -27922.567} C_VEL
LIN {X 0,Y 161.731,Z 880.534,A -85,B 0,C 180,E1 -27929.643,E2 -27929.643} C_VEL
LIN {X 0,Y 176.432,Z 876.109,A -85,B 0,C 180,E1 -27936.114,E2 -27936.114} C_VEL
LIN {X 0,Y 187.683,Z 872.879,A -85,B 0,C 180,E1 -27939.769,E2 -27939.769} C_VEL
LIN {X 0,Y 175.991,Z 883.431,A -85,B 0,C 180,E1 -27944.79,E2 -27944.79} C_VEL
LIN {X 0,Y 165.356,Z 892.3,A -85,B 0,C 180,E1 -27950.585,E2 -27950.585} C_VEL
LIN {X 0,Y 155.917,Z 899.704,A -85,B 0,C 180,E1 -27957.405,E2 -27957.405} C_VEL
LIN {X 0,Y 148.567,Z 905.284,A -85,B 0,C 180,E1 -27964.912,E2 -27964.912} C_VEL
LIN {X 0,Y 143.438,Z 909.177,A -85,B 0,C 180,E1 -27972.975,E2 -27972.975} C_VEL
LIN {X 0,Y 140.551,Z 911.477,A -85,B 0,C 180,E1 -27981.44,E2 -27981.44} C_VEL
LIN {X 0,Y 139.664,Z 912.242,A -85,B 0,C 180,E1 -27990,E2 -27990} C_VEL
LIN {X 0,Y 140.511,Z 911.519,A -85,B 0,C 180,E1 -27998.45,E2 -27998.45} C_VEL
LIN {X 0,Y 143.212,Z 909.371,A -85,B 0,C 180,E1 -28006.634,E2 -28006.634} C_VEL
LIN {X 0,Y 148.213,Z 905.599,A -85,B 0,C 180,E1 -28014.725,E2 -28014.725} C_VEL
LIN {X 0,Y 155.445,Z 900.141,A -85,B 0,C 180,E1 -28022.269,E2 -28022.269} C_VEL
LIN {X 0,Y 164.776,Z 892.87,A -85,B 0,C 180,E1 -28029.13,E2 -28029.13} C_VEL
LIN {X 0,Y 175.515,Z 883.986,A -85,B 0,C 180,E1 -28035.056,E2 -28035.056} C_VEL
LIN {X 0,Y 186.777,Z 873.9,A -85,B 0,C 180,E1 -28039.954,E2 -28039.954} C_VEL
LIN {X 0,Y 198.583,Z 862.311,A -85,B 0,C 180,E1 -28044.16,E2 -28044.16} C_VEL
LIN {X 0,Y 210.497,Z 849.365,A -85,B 0,C 180,E1 -28047.728,E2 -28047.728} C_VEL
LIN {X 0,Y 222.278,Z 835.044,A -85,B 0,C 180,E1 -28050.772,E2 -28050.772} C_VEL
LIN {X 0,Y 233.356,Z 819.821,A -85,B 0,C 180,E1 -28053.302,E2 -28053.302} C_VEL
LIN {X 0,Y 243.96,Z 803.186,A -85,B 0,C 180,E1 -28055.489,E2 -28055.489} C_VEL
LIN {X 0,Y 253.795,Z 785.269,A -85,B 0,C 180,E1 -28057.362,E2 -28057.362} C_VEL
LIN {X 0,Y 262.516,Z 766.436,A -85,B 0,C 180,E1 -28058.935,E2 -28058.935} C_VEL
LIN {X 0,Y 270.115,Z 746.368,A -85,B 0,C 180,E1 -28060.263,E2 -28060.263} C_VEL
LIN {X 0,Y 276.439,Z 725.063,A -85,B 0,C 180,E1 -28061.381,E2 -28061.381} C_VEL
LIN {X 0,Y 286.276,Z 686.048,A -85,B 0,C 180,E1 -28062.963,E2 -28062.963} C_VEL
LIN {X 0,Y 295.1,Z 647.201,A -85,B 0,C 180,E1 -28064.124,E2 -28064.124} C_VEL
LIN {X 0,Y 303.348,Z 604.971,A -85,B 0,C 180,E1 -28065.036,E2 -28065.036} C_VEL
LIN {X 0,Y 309.935,Z 562.716,A -85,B 0,C 180,E1 -28065.802,E2 -28065.802} C_VEL
LIN {X 0,Y 316.767,Z 503.485,A -85,B 0,C 180,E1 -28066.718,E2 -28066.718} C_VEL
LIN {X 0,Y 318.692,Z 488.261,A -85,B 0,C 180,E1 -28066.953,E2 -28066.953} C_VEL
LIN {X 0,Y 319.062,Z 486.716,A -85,B 0,C 180,E1 -28067.006,E2 -28067.006} C_VEL
LIN {X 0,Y 318.382,Z 479.662,A -85,B 0,C 180,E1 -28070.145,E2 -28070.145} C_VEL
LIN {X 0,Y 318.091,Z 474.647,A -85,B 0,C 180,E1 -28073.14,E2 -28073.14} C_VEL
LIN {X 0,Y 318.171,Z 471.916,A -85,B 0,C 180,E1 -28075.494,E2 -28075.494} C_VEL
LIN {X 0,Y 318.595,Z 469.461,A -85,B 0,C 180,E1 -28078.381,E2 -28078.381} C_VEL
LIN {X 0,Y 319.79,Z 469.035,A -85,B 0,C 180,E1 -28082.374,E2 -28082.374} C_VEL
LIN {X 0,Y 319.391,Z 477.958,A -85,B 0,C 180,E1 -28085.299,E2 -28085.299} C_VEL
LIN {X 0,Y 319.36,Z 481.29,A -85,B 0,C 180,E1 -28086.245,E2 -28086.245} C_VEL
LIN {X 0,Y 308.857,Z 531.488,A -85,B 0,C 180,E1 -28087.318,E2 -28087.318} C_VEL
LIN {X 0,Y 304.602,Z 570.726,A -85,B 0,C 180,E1 -28088.063,E2 -28088.063} C_VEL
LIN {X 0,Y 303.584,Z 578.422,A -85,B 0,C 180,E1 -28088.022,E2 -28088.022} C_VEL
LIN {X 0,Y 299.983,Z 598.958,A -85,B 0,C 180,E1 -28087.228,E2 -28087.228} C_VEL
LIN {X 0,Y 298.908,Z 605.538,A -85,B 0,C 180,E1 -28087.217,E2 -28087.217} C_VEL
LIN {X 0,Y 292.126,Z 644.737,A -85,B 0,C 180,E1 -28087.959,E2 -28087.959} C_VEL
LIN {X 0,Y 283.674,Z 683.502,A -85,B 0,C 180,E1 -28088.856,E2 -28088.856} C_VEL
LIN {X 0,Y 274.58,Z 718.346,A -85,B 0,C 180,E1 -28089.855,E2 -28089.855} C_VEL
LIN {X 0,Y 265.214,Z 749.721,A -85,B 0,C 180,E1 -28090.999,E2 -28090.999} C_VEL
LIN {X 0,Y 256.749,Z 774.715,A -85,B 0,C 180,E1 -28092.177,E2 -28092.177} C_VEL
LIN {X 0,Y 248.354,Z 794.709,A -85,B 0,C 180,E1 -28093.38,E2 -28093.38} C_VEL
LIN {X 0,Y 238.929,Z 813.466,A -85,B 0,C 180,E1 -28094.826,E2 -28094.826} C_VEL
LIN {X 0,Y 227.892,Z 832.166,A -85,B 0,C 180,E1 -28096.673,E2 -28096.673} C_VEL
LIN {X 0,Y 215.73,Z 850.037,A -85,B 0,C 180,E1 -28099,E2 -28099} C_VEL
LIN {X 0,Y 203.452,Z 865.975,A -85,B 0,C 180,E1 -28101.742,E2 -28101.742} C_VEL
LIN {X 0,Y 190.921,Z 880.546,A -85,B 0,C 180,E1 -28105.038,E2 -28105.038} C_VEL
LIN {X 0,Y 177.634,Z 894.634,A -85,B 0,C 180,E1 -28109.322,E2 -28109.322} C_VEL
LIN {X 0,Y 165.007,Z 906.981,A -85,B 0,C 180,E1 -28114.501,E2 -28114.501} C_VEL
LIN {X 0,Y 153.681,Z 917.511,A -85,B 0,C 180,E1 -28120.589,E2 -28120.589} C_VEL
LIN {X 0,Y 143.666,Z 926.783,A -85,B 0,C 180,E1 -28128.077,E2 -28128.077} C_VEL
LIN {X 0,Y 136.167,Z 934.249,A -85,B 0,C 180,E1 -28136.583,E2 -28136.583} C_VEL
LIN {X 0,Y 131.636,Z 939.904,A -85,B 0,C 180,E1 -28145.784,E2 -28145.784} C_VEL
LIN {X 0,Y 130.073,Z 943.825,A -85,B 0,C 180,E1 -28155.305,E2 -28155.305} C_VEL
LIN {X 0,Y 130.754,Z 945.872,A -85,B 0,C 180,E1 -28163.854,E2 -28163.854} C_VEL
LIN {X 0,Y 131.553,Z 946.403,A -85,B 0,C 180,E1 -28169.129,E2 -28169.129} C_VEL
LIN {X 0,Y 131.255,Z 946.219,A -85,B 0,C 180,E1 -28173.664,E2 -28173.664} C_VEL
LIN {X 0,Y 130.432,Z 944.755,A -85,B 0,C 180,E1 -28181.497,E2 -28181.497} C_VEL
LIN {X 0,Y 131.622,Z 941.268,A -85,B 0,C 180,E1 -28191.386,E2 -28191.386} C_VEL
LIN {X 0,Y 136.128,Z 936.145,A -85,B 0,C 180,E1 -28200.942,E2 -28200.942} C_VEL
LIN {X 0,Y 150.072,Z 934.581,A -85,B 0,C 180,E1 -28215.606,E2 -28215.606} C_VEL
LIN {X 0,Y 163.874,Z 932.543,A -85,B 0,C 180,E1 -28223.534,E2 -28223.534} C_VEL
LIN {X 0,Y 150.837,Z 926.373,A -85,B 0,C 180,E1 -28230.624,E2 -28230.624} C_VEL
LIN {X 0,Y 141.01,Z 918.536,A -85,B 0,C 180,E1 -28238.799,E2 -28238.799} C_VEL
LIN {X 0,Y 134.919,Z 909.631,A -85,B 0,C 180,E1 -28247.154,E2 -28247.154} C_VEL
LIN {X 0,Y 131.698,Z 899.21,A -85,B 0,C 180,E1 -28255.646,E2 -28255.646} C_VEL
LIN {X 0,Y 131.396,Z 897.616,A -85,B 0,C 180,E1 -28256.947,E2 -28256.947} C_VEL
LIN {X 0,Y 131.291,Z 896.368,A -85,B 0,C 180,E1 -28260.873,E2 -28260.873} C_VEL
LIN {X 0,Y 131.636,Z 895.609,A -85,B 0,C 180,E1 -28263.048,E2 -28263.048} C_VEL
LIN {X 0,Y 133.054,Z 893.881,A -85,B 0,C 180,E1 -28268.209,E2 -28268.209} C_VEL
LIN {X 0,Y 145.133,Z 887.999,A -85,B 0,C 180,E1 -28283.984,E2 -28283.984} C_VEL
LIN {X 0,Y 160.953,Z 883.121,A -85,B 0,C 180,E1 -28293.566,E2 -28293.566} C_VEL
LIN {X 0,Y 177.556,Z 878.499,A -85,B 0,C 180,E1 -28299.824,E2 -28299.824} C_VEL
LIN {X 0,Y 165.266,Z 888.707,A -85,B 0,C 180,E1 -28305.426,E2 -28305.426} C_VEL
LIN {X 0,Y 154.247,Z 897.11,A -85,B 0,C 180,E1 -28311.987,E2 -28311.987} C_VEL
LIN {X 0,Y 145.127,Z 903.677,A -85,B 0,C 180,E1 -28319.455,E2 -28319.455} C_VEL
LIN {X 0,Y 138.174,Z 908.541,A -85,B 0,C 180,E1 -28327.895,E2 -28327.895} C_VEL
LIN {X 0,Y 133.91,Z 911.574,A -85,B 0,C 180,E1 -28336.616,E2 -28336.616} C_VEL
LIN {X 0,Y 131.939,Z 913.06,A -85,B 0,C 180,E1 -28345.653,E2 -28345.653} C_VEL
LIN {X 0,Y 131.929,Z 913.069,A -85,B 0,C 180,E1 -28354.346,E2 -28354.346} C_VEL
LIN {X 0,Y 133.738,Z 911.71,A -85,B 0,C 180,E1 -28362.961,E2 -28362.961} C_VEL
LIN {X 0,Y 137.866,Z 908.793,A -85,B 0,C 180,E1 -28371.708,E2 -28371.708} C_VEL
LIN {X 0,Y 144.406,Z 904.245,A -85,B 0,C 180,E1 -28379.903,E2 -28379.903} C_VEL
LIN {X 0,Y 153.219,Z 897.953,A -85,B 0,C 180,E1 -28387.366,E2 -28387.366} C_VEL
LIN {X 0,Y 163.489,Z 890.199,A -85,B 0,C 180,E1 -28393.717,E2 -28393.717} C_VEL
LIN {X 0,Y 174.695,Z 881.086,A -85,B 0,C 180,E1 -28399.07,E2 -28399.07} C_VEL
LIN {X 0,Y 186.416,Z 870.683,A -85,B 0,C 180,E1 -28403.568,E2 -28403.568} C_VEL
LIN {X 0,Y 199.022,Z 858.306,A -85,B 0,C 180,E1 -28407.569,E2 -28407.569} C_VEL
LIN {X 0,Y 211.613,Z 844.474,A -85,B 0,C 180,E1 -28410.943,E2 -28410.943} C_VEL
LIN {X 0,Y 223.463,Z 829.758,A -85,B 0,C 180,E1 -28413.706,E2 -28413.706} C_VEL
LIN {X 0,Y 234.704,Z 813.874,A -85,B 0,C 180,E1 -28416.038,E2 -28416.038} C_VEL
LIN {X 0,Y 245.275,Z 796.649,A -85,B 0,C 180,E1 -28418.037,E2 -28418.037} C_VEL
LIN {X 0,Y 254.773,Z 778.488,A -85,B 0,C 180,E1 -28419.716,E2 -28419.716} C_VEL
LIN {X 0,Y 263.118,Z 759.391,A -85,B 0,C 180,E1 -28421.127,E2 -28421.127} C_VEL
LIN {X 0,Y 270.288,Z 739.093,A -85,B 0,C 180,E1 -28422.32,E2 -28422.32} C_VEL
LIN {X 0,Y 279.287,Z 706.135,A -85,B 0,C 180,E1 -28423.798,E2 -28423.798} C_VEL
LIN {X 0,Y 288.343,Z 669.322,A -85,B 0,C 180,E1 -28425.059,E2 -28425.059} C_VEL
LIN {X 0,Y 296.706,Z 630.979,A -85,B 0,C 180,E1 -28426.01,E2 -28426.01} C_VEL
LIN {X 0,Y 304.282,Z 589.346,A -85,B 0,C 180,E1 -28426.805,E2 -28426.805} C_VEL
LIN {X 0,Y 310.403,Z 545.763,A -85,B 0,C 180,E1 -28427.517,E2 -28427.517} C_VEL
LIN {X 0,Y 316.559,Z 491.823,A -85,B 0,C 180,E1 -28428.337,E2 -28428.337} C_VEL
LIN {X 0,Y 316.136,Z 485.383,A -85,B 0,C 180,E1 -28431.451,E2 -28431.451} C_VEL
LIN {X 0,Y 316.087,Z 481.274,A -85,B 0,C 180,E1 -28434.19,E2 -28434.19} C_VEL
LIN {X 0,Y 316.278,Z 479.178,A -85,B 0,C 180,E1 -28436.193,E2 -28436.193} C_VEL
LIN {X 0,Y 316.762,Z 477.214,A -85,B 0,C 180,E1 -28438.553,E2 -28438.553} C_VEL
LIN {X 0,Y 317.777,Z 476.774,A -85,B 0,C 180,E1 -28442.029,E2 -28442.029} C_VEL
LIN {X 0,Y 317.328,Z 485.126,A -85,B 0,C 180,E1 -28444.745,E2 -28444.745} C_VEL
LIN {X 0,Y 317.251,Z 485.961,A -85,B 0,C 180,E1 -28444.907,E2 -28444.907} C_VEL
LIN {X 0,Y 308.165,Z 528.507,A -85,B 0,C 180,E1 -28445.781,E2 -28445.781} C_VEL
LIN {X 0,Y 300.294,Z 596.054,A -85,B 0,C 180,E1 -28447.041,E2 -28447.041} C_VEL
LIN {X 0,Y 298.908,Z 605.538,A -85,B 0,C 180,E1 -28447.217,E2 -28447.217} C_VEL
LIN {X 0,Y 297.623,Z 613.185,A -85,B 0,C 180,E1 -28447.166,E2 -28447.166} C_VEL
LIN {X 0,Y 293.15,Z 633.523,A -85,B 0,C 180,E1 -28446.332,E2 -28446.332} C_VEL
LIN {X 0,Y 291.743,Z 640.045,A -85,B 0,C 180,E1 -28446.314,E2 -28446.314} C_VEL
LIN {X 0,Y 283.564,Z 677.85,A -85,B 0,C 180,E1 -28447.123,E2 -28447.123} C_VEL
LIN {X 0,Y 274.075,Z 714.312,A -85,B 0,C 180,E1 -28448.085,E2 -28448.085} C_VEL
LIN {X 0,Y 264.128,Z 747.376,A -85,B 0,C 180,E1 -28449.212,E2 -28449.212} C_VEL
LIN {X 0,Y 255.598,Z 772.323,A -85,B 0,C 180,E1 -28450.309,E2 -28450.309} C_VEL
LIN {X 0,Y 247.216,Z 792.135,A -85,B 0,C 180,E1 -28451.431,E2 -28451.431} C_VEL
LIN {X 0,Y 237.839,Z 810.619,A -85,B 0,C 180,E1 -28452.751,E2 -28452.751} C_VEL
LIN {X 0,Y 227.114,Z 828.659,A -85,B 0,C 180,E1 -28454.403,E2 -28454.403} C_VEL
LIN {X 0,Y 215.477,Z 845.69,A -85,B 0,C 180,E1 -28456.443,E2 -28456.443} C_VEL
LIN {X 0,Y 202.861,Z 861.92,A -85,B 0,C 180,E1 -28458.984,E2 -28458.984} C_VEL
LIN {X 0,Y 189.092,Z 877.629,A -85,B 0,C 180,E1 -28462.275,E2 -28462.275} C_VEL
LIN {X 0,Y 175.969,Z 891.153,A -85,B 0,C 180,E1 -28466.132,E2 -28466.132} C_VEL
LIN {X 0,Y 163.071,Z 903.351,A -85,B 0,C 180,E1 -28470.86,E2 -28470.86} C_VEL
LIN {X 0,Y 150.851,Z 914.202,A -85,B 0,C 180,E1 -28476.676,E2 -28476.676} C_VEL
LIN {X 0,Y 139.642,Z 923.886,A -85,B 0,C 180,E1 -28483.992,E2 -28483.992} C_VEL
LIN {X 0,Y 130.601,Z 931.904,A -85,B 0,C 180,E1 -28492.784,E2 -28492.784} C_VEL
LIN {X 0,Y 124.836,Z 937.897,A -85,B 0,C 180,E1 -28502.319,E2 -28502.319} C_VEL
LIN {X 0,Y 122.274,Z 942.151,A -85,B 0,C 180,E1 -28512.389,E2 -28512.389} C_VEL
LIN {X 0,Y 122.512,Z 944.619,A -85,B 0,C 180,E1 -28522.025,E2 -28522.025} C_VEL
LIN {X 0,Y 123.554,Z 945.374,A -85,B 0,C 180,E1 -28528.609,E2 -28528.609} C_VEL
LIN {X 0,Y 123.482,Z 945.318,A -85,B 0,C 180,E1 -28532.321,E2 -28532.321} C_VEL
LIN {X 0,Y 122.538,Z 944.296,A -85,B 0,C 180,E1 -28539.867,E2 -28539.867} C_VEL
LIN {X 0,Y 123.22,Z 941.367,A -85,B 0,C 180,E1 -28549.927,E2 -28549.927} C_VEL
LIN {X 0,Y 127.422,Z 936.412,A -85,B 0,C 180,E1 -28560.324,E2 -28560.324} C_VEL
LIN {X 0,Y 130.796,Z 933.61,A -85,B 0,C 180,E1 -28564.985,E2 -28564.985} C_VEL
LIN {X 0,Y 146.55,Z 932.224,A -85,B 0,C 180,E1 -28579.23,E2 -28579.23} C_VEL
LIN {X 0,Y 153.997,Z 931.267,A -85,B 0,C 180,E1 -28583.419,E2 -28583.419} C_VEL
LIN {X 0,Y 140.918,Z 924.181,A -85,B 0,C 180,E1 -28591.151,E2 -28591.151} C_VEL
LIN {X 0,Y 131.806,Z 915.915,A -85,B 0,C 180,E1 -28599.576,E2 -28599.576} C_VEL
LIN {X 0,Y 126.086,Z 906.158,A -85,B 0,C 180,E1 -28608.565,E2 -28608.565} C_VEL
LIN {X 0,Y 124.965,Z 903.28,A -85,B 0,C 180,E1 -28611.256,E2 -28611.256} C_VEL
LIN {X 0,Y 124.169,Z 901.608,A -85,B 0,C 180,E1 -28616.306,E2 -28616.306} C_VEL
LIN {X 0,Y 124.649,Z 899.12,A -85,B 0,C 180,E1 -28624.14,E2 -28624.14} C_VEL
LIN {X 0,Y 126.324,Z 897.358,A -85,B 0,C 180,E1 -28629.568,E2 -28629.568} C_VEL
LIN {X 0,Y 143.508,Z 890.285,A -85,B 0,C 180,E1 -28648.735,E2 -28648.735} C_VEL
LIN {X 0,Y 163.76,Z 884.642,A -85,B 0,C 180,E1 -28658.521,E2 -28658.521} C_VEL
LIN {X 0,Y 167.509,Z 883.655,A -85,B 0,C 180,E1 -28659.824,E2 -28659.824} C_VEL
LIN {X 0,Y 155.027,Z 893.177,A -85,B 0,C 180,E1 -28665.846,E2 -28665.846} C_VEL
LIN {X 0,Y 144.113,Z 900.842,A -85,B 0,C 180,E1 -28672.87,E2 -28672.87} C_VEL
LIN {X 0,Y 134.985,Z 906.898,A -85,B 0,C 180,E1 -28681.217,E2 -28681.217} C_VEL
LIN {X 0,Y 128.518,Z 911.072,A -85,B 0,C 180,E1 -28690.455,E2 -28690.455} C_VEL
LIN {X 0,Y 124.863,Z 913.482,A -85,B 0,C 180,E1 -28700.318,E2 -28700.318} C_VEL
LIN {X 0,Y 123.789,Z 914.243,A -85,B 0,C 180,E1 -28710,E2 -28710} C_VEL
LIN {X 0,Y 124.741,Z 913.563,A -85,B 0,C 180,E1 -28719.225,E2 -28719.225} C_VEL
LIN {X 0,Y 128.027,Z 911.398,A -85,B 0,C 180,E1 -28728.675,E2 -28728.675} C_VEL
LIN {X 0,Y 133.884,Z 907.644,A -85,B 0,C 180,E1 -28737.583,E2 -28737.583} C_VEL
LIN {X 0,Y 142.191,Z 902.207,A -85,B 0,C 180,E1 -28745.708,E2 -28745.708} C_VEL
LIN {X 0,Y 152.27,Z 895.265,A -85,B 0,C 180,E1 -28752.654,E2 -28752.654} C_VEL
LIN {X 0,Y 163.846,Z 886.686,A -85,B 0,C 180,E1 -28758.644,E2 -28758.644} C_VEL
LIN {X 0,Y 176.249,Z 876.617,A -85,B 0,C 180,E1 -28763.667,E2 -28763.667} C_VEL
LIN {X 0,Y 188.963,Z 865.176,A -85,B 0,C 180,E1 -28767.847,E2 -28767.847} C_VEL
LIN {X 0,Y 201.681,Z 852.388,A -85,B 0,C 180,E1 -28771.345,E2 -28771.345} C_VEL
LIN {X 0,Y 214.17,Z 838.231,A -85,B 0,C 180,E1 -28774.297,E2 -28774.297} C_VEL
LIN {X 0,Y 226.259,Z 822.637,A -85,B 0,C 180,E1 -28776.809,E2 -28776.809} C_VEL
LIN {X 0,Y 237.401,Z 806.096,A -85,B 0,C 180,E1 -28778.894,E2 -28778.894} C_VEL
LIN {X 0,Y 247.9,Z 787.962,A -85,B 0,C 180,E1 -28780.704,E2 -28780.704} C_VEL
LIN {X 0,Y 257.242,Z 768.611,A -85,B 0,C 180,E1 -28782.233,E2 -28782.233} C_VEL
LIN {X 0,Y 264.943,Z 749.12,A -85,B 0,C 180,E1 -28783.454,E2 -28783.454} C_VEL
LIN {X 0,Y 271.413,Z 728.406,A -85,B 0,C 180,E1 -28784.493,E2 -28784.493} C_VEL
LIN {X 0,Y 281.158,Z 691.859,A -85,B 0,C 180,E1 -28785.927,E2 -28785.927} C_VEL
LIN {X 0,Y 289.738,Z 656.317,A -85,B 0,C 180,E1 -28786.973,E2 -28786.973} C_VEL
LIN {X 0,Y 297.75,Z 618.076,A -85,B 0,C 180,E1 -28787.78,E2 -28787.78} C_VEL
LIN {X 0,Y 304.748,Z 576.937,A -85,B 0,C 180,E1 -28788.497,E2 -28788.497} C_VEL
LIN {X 0,Y 310.385,Z 533.116,A -85,B 0,C 180,E1 -28789.157,E2 -28789.157} C_VEL
LIN {X 0,Y 314.378,Z 497.094,A -85,B 0,C 180,E1 -28789.689,E2 -28789.689} C_VEL
LIN {X 0,Y 314.045,Z 491.397,A -85,B 0,C 180,E1 -28792.683,E2 -28792.683} C_VEL
LIN {X 0,Y 314.25,Z 487.496,A -85,B 0,C 180,E1 -28795.62,E2 -28795.62} C_VEL
LIN {X 0,Y 314.958,Z 484.973,A -85,B 0,C 180,E1 -28798.727,E2 -28798.727} C_VEL
LIN {X 0,Y 315.776,Z 484.695,A -85,B 0,C 180,E1 -28801.724,E2 -28801.724} C_VEL
LIN {X 0,Y 315.345,Z 490.279,A -85,B 0,C 180,E1 -28803.548,E2 -28803.548} C_VEL
LIN {X 0,Y 307.685,Z 525.621,A -85,B 0,C 180,E1 -28804.241,E2 -28804.241} C_VEL
LIN {X 0,Y 299.585,Z 593.552,A -85,B 0,C 180,E1 -28805.478,E2 -28805.478} C_VEL
LIN {X 0,Y 293.231,Z 632.503,A -85,B 0,C 180,E1 -28806.175,E2 -28806.175} C_VEL
LIN {X 0,Y 291.743,Z 640.045,A -85,B 0,C 180,E1 -28806.314,E2 -28806.314} C_VEL
LIN {X 0,Y 290.098,Z 647.63,A -85,B 0,C 180,E1 -28806.254,E2 -28806.254} C_VEL
LIN {X 0,Y 284.562,Z 668.867,A -85,B 0,C 180,E1 -28805.413,E2 -28805.413} C_VEL
LIN {X 0,Y 283.18,Z 674.24,A -85,B 0,C 180,E1 -28805.438,E2 -28805.438} C_VEL
LIN {X 0,Y 273.552,Z 711.211,A -85,B 0,C 180,E1 -28806.346,E2 -28806.346} C_VEL
LIN {X 0,Y 262.941,Z 746.099,A -85,B 0,C 180,E1 -28807.45,E2 -28807.45} C_VEL
LIN {X 0,Y 254.254,Z 771.078,A -85,B 0,C 180,E1 -28808.483,E2 -28808.483} C_VEL
LIN {X 0,Y 245.865,Z 790.576,A -85,B 0,C 180,E1 -28809.528,E2 -28809.528} C_VEL
LIN {X 0,Y 236.148,Z 809.356,A -85,B 0,C 180,E1 -28810.788,E2 -28810.788} C_VEL
LIN {X 0,Y 225.191,Z 827.407,A -85,B 0,C 180,E1 -28812.355,E2 -28812.355} C_VEL
LIN {X 0,Y 213.547,Z 844.088,A -85,B 0,C 180,E1 -28814.249,E2 -28814.249} C_VEL
LIN {X 0,Y 200.977,Z 859.884,A -85,B 0,C 180,E1 -28816.572,E2 -28816.572} C_VEL
LIN {X 0,Y 186.892,Z 875.571,A -85,B 0,C 180,E1 -28819.675,E2 -28819.675} C_VEL
LIN {X 0,Y 172.606,Z 889.815,A -85,B 0,C 180,E1 -28823.56,E2 -28823.56} C_VEL
LIN {X 0,Y 158.904,Z 902.205,A -85,B 0,C 180,E1 -28828.245,E2 -28828.245} C_VEL
LIN {X 0,Y 145.971,Z 913.076,A -85,B 0,C 180,E1 -28834.02,E2 -28834.02} C_VEL
LIN {X 0,Y 134.202,Z 922.546,A -85,B 0,C 180,E1 -28841.192,E2 -28841.192} C_VEL
LIN {X 0,Y 124.409,Z 930.496,A -85,B 0,C 180,E1 -28849.987,E2 -28849.987} C_VEL
LIN {X 0,Y 117.675,Z 936.658,A -85,B 0,C 180,E1 -28860.078,E2 -28860.078} C_VEL
LIN {X 0,Y 114.432,Z 941.1,A -85,B 0,C 180,E1 -28871.138,E2 -28871.138} C_VEL
LIN {X 0,Y 114.474,Z 943.592,A -85,B 0,C 180,E1 -28881.461,E2 -28881.461} C_VEL
LIN {X 0,Y 115.589,Z 944.369,A -85,B 0,C 180,E1 -28888.513,E2 -28888.513} C_VEL
LIN {X 0,Y 115.509,Z 944.312,A -85,B 0,C 180,E1 -28892.481,E2 -28892.481} C_VEL
LIN {X 0,Y 114.53,Z 943.156,A -85,B 0,C 180,E1 -28901.074,E2 -28901.074} C_VEL
LIN {X 0,Y 115.655,Z 940.131,A -85,B 0,C 180,E1 -28911.824,E2 -28911.824} C_VEL
LIN {X 0,Y 120.599,Z 935.16,A -85,B 0,C 180,E1 -28922.61,E2 -28922.61} C_VEL
LIN {X 0,Y 126.155,Z 930.988,A -85,B 0,C 180,E1 -28929.352,E2 -28929.352} C_VEL
LIN {X 0,Y 143.23,Z 929.701,A -85,B 0,C 180,E1 -28942.735,E2 -28942.735} C_VEL
LIN {X 0,Y 144.045,Z 929.534,A -85,B 0,C 180,E1 -28943.347,E2 -28943.347} C_VEL
LIN {X 0,Y 131.517,Z 921.923,A -85,B 0,C 180,E1 -28951.382,E2 -28951.382} C_VEL
LIN {X 0,Y 122.649,Z 912.864,A -85,B 0,C 180,E1 -28960.473,E2 -28960.473} C_VEL
LIN {X 0,Y 119.971,Z 908.753,A -85,B 0,C 180,E1 -28964.532,E2 -28964.532} C_VEL
LIN {X 0,Y 117.846,Z 906.924,A -85,B 0,C 180,E1 -28970.23,E2 -28970.23} C_VEL
LIN {X 0,Y 116.77,Z 904.113,A -85,B 0,C 180,E1 -28979.509,E2 -28979.509} C_VEL
LIN {X 0,Y 117.529,Z 902.473,A -85,B 0,C 180,E1 -28984.88,E2 -28984.88} C_VEL
LIN {X 0,Y 137.218,Z 893.895,A -85,B 0,C 180,E1 -29010.185,E2 -29010.185} C_VEL
LIN {X 0,Y 157.255,Z 888.639,A -85,B 0,C 180,E1 -29019.895,E2 -29019.895} C_VEL
LIN {X 0,Y 144.759,Z 897.353,A -85,B 0,C 180,E1 -29026.312,E2 -29026.312} C_VEL
LIN {X 0,Y 133.967,Z 904.276,A -85,B 0,C 180,E1 -29033.869,E2 -29033.869} C_VEL
LIN {X 0,Y 125.152,Z 909.614,A -85,B 0,C 180,E1 -29042.909,E2 -29042.909} C_VEL
LIN {X 0,Y 119.428,Z 912.999,A -85,B 0,C 180,E1 -29052.458,E2 -29052.458} C_VEL
LIN {X 0,Y 116.437,Z 914.813,A -85,B 0,C 180,E1 -29062.599,E2 -29062.599} C_VEL
LIN {X 0,Y 115.901,Z 915.159,A -85,B 0,C 180,E1 -29072.472,E2 -29072.472} C_VEL
LIN {X 0,Y 117.515,Z 914.184,A -85,B 0,C 180,E1 -29082.281,E2 -29082.281} C_VEL
LIN {X 0,Y 121.768,Z 911.67,A -85,B 0,C 180,E1 -29092.193,E2 -29092.193} C_VEL
LIN {X 0,Y 128.759,Z 907.546,A -85,B 0,C 180,E1 -29101.352,E2 -29101.352} C_VEL
LIN {X 0,Y 138.261,Z 901.699,A -85,B 0,C 180,E1 -29109.524,E2 -29109.524} C_VEL
LIN {X 0,Y 149.737,Z 894.118,A -85,B 0,C 180,E1 -29116.544,E2 -29116.544} C_VEL
LIN {X 0,Y 161.984,Z 885.293,A -85,B 0,C 180,E1 -29122.196,E2 -29122.196} C_VEL
LIN {X 0,Y 175.23,Z 874.715,A -85,B 0,C 180,E1 -29127.014,E2 -29127.014} C_VEL
LIN {X 0,Y 188.65,Z 862.724,A -85,B 0,C 180,E1 -29130.99,E2 -29130.99} C_VEL
LIN {X 0,Y 201.959,Z 849.303,A -85,B 0,C 180,E1 -29134.299,E2 -29134.299} C_VEL
LIN {X 0,Y 214.942,Z 834.399,A -85,B 0,C 180,E1 -29137.084,E2 -29137.084} C_VEL
LIN {X 0,Y 226.972,Z 818.579,A -85,B 0,C 180,E1 -29139.364,E2 -29139.364} C_VEL
LIN {X 0,Y 238.077,Z 801.689,A -85,B 0,C 180,E1 -29141.275,E2 -29141.275} C_VEL
LIN {X 0,Y 247.55,Z 784.883,A -85,B 0,C 180,E1 -29142.796,E2 -29142.796} C_VEL
LIN {X 0,Y 256.113,Z 766.908,A -85,B 0,C 180,E1 -29144.113,E2 -29144.113} C_VEL
LIN {X 0,Y 263.228,Z 748.875,A -85,B 0,C 180,E1 -29145.18,E2 -29145.18} C_VEL
LIN {X 0,Y 269.781,Z 728.009,A -85,B 0,C 180,E1 -29146.18,E2 -29146.18} C_VEL
LIN {X 0,Y 279.027,Z 694.221,A -85,B 0,C 180,E1 -29147.465,E2 -29147.465} C_VEL
LIN {X 0,Y 287.478,Z 660.233,A -85,B 0,C 180,E1 -29148.446,E2 -29148.446} C_VEL
LIN {X 0,Y 295.644,Z 622.289,A -85,B 0,C 180,E1 -29149.23,E2 -29149.23} C_VEL
LIN {X 0,Y 302.903,Z 580.645,A -85,B 0,C 180,E1 -29149.93,E2 -29149.93} C_VEL
LIN {X 0,Y 308.599,Z 537.418,A -85,B 0,C 180,E1 -29150.56,E2 -29150.56} C_VEL
LIN {X 0,Y 312.519,Z 502.545,A -85,B 0,C 180,E1 -29151.073,E2 -29151.073} C_VEL
LIN {X 0,Y 312.032,Z 498.801,A -85,B 0,C 180,E1 -29153.098,E2 -29153.098} C_VEL
LIN {X 0,Y 312.365,Z 495.078,A -85,B 0,C 180,E1 -29155.962,E2 -29155.962} C_VEL
LIN {X 0,Y 313.051,Z 492.707,A -85,B 0,C 180,E1 -29158.902,E2 -29158.902} C_VEL
LIN {X 0,Y 313.821,Z 492.476,A -85,B 0,C 180,E1 -29161.369,E2 -29161.369} C_VEL
LIN {X 0,Y 313.536,Z 495.061,A -85,B 0,C 180,E1 -29162.18,E2 -29162.18} C_VEL
LIN {X 0,Y 307.401,Z 522.954,A -85,B 0,C 180,E1 -29162.701,E2 -29162.701} C_VEL
LIN {X 0,Y 299.158,Z 590.648,A -85,B 0,C 180,E1 -29163.896,E2 -29163.896} C_VEL
LIN {X 0,Y 292.682,Z 629.917,A -85,B 0,C 180,E1 -29164.575,E2 -29164.575} C_VEL
LIN {X 0,Y 284.385,Z 669.361,A -85,B 0,C 180,E1 -29165.329,E2 -29165.329} C_VEL
LIN {X 0,Y 283.18,Z 674.24,A -85,B 0,C 180,E1 -29165.438,E2 -29165.438} C_VEL
LIN {X 0,Y 281.194,Z 681.746,A -85,B 0,C 180,E1 -29165.408,E2 -29165.408} C_VEL
LIN {X 0,Y 275.209,Z 701.747,A -85,B 0,C 180,E1 -29164.607,E2 -29164.607} C_VEL
LIN {X 0,Y 273.269,Z 708.115,A -85,B 0,C 180,E1 -29164.603,E2 -29164.603} C_VEL
LIN {X 0,Y 262.244,Z 744.106,A -85,B 0,C 180,E1 -29165.647,E2 -29165.647} C_VEL
LIN {X 0,Y 253.647,Z 768.686,A -85,B 0,C 180,E1 -29166.588,E2 -29166.588} C_VEL
LIN {X 0,Y 245.11,Z 788.404,A -85,B 0,C 180,E1 -29167.571,E2 -29167.571} C_VEL
LIN {X 0,Y 235.208,Z 807.344,A -85,B 0,C 180,E1 -29168.744,E2 -29168.744} C_VEL
LIN {X 0,Y 223.563,Z 826.196,A -85,B 0,C 180,E1 -29170.279,E2 -29170.279} C_VEL
LIN {X 0,Y 211.318,Z 843.293,A -85,B 0,C 180,E1 -29172.114,E2 -29172.114} C_VEL
LIN {X 0,Y 197.751,Z 859.805,A -85,B 0,C 180,E1 -29174.443,E2 -29174.443} C_VEL
LIN {X 0,Y 184.234,Z 874.362,A -85,B 0,C 180,E1 -29177.215,E2 -29177.215} C_VEL
LIN {X 0,Y 170.038,Z 888.064,A -85,B 0,C 180,E1 -29180.775,E2 -29180.775} C_VEL
LIN {X 0,Y 155.84,Z 900.418,A -85,B 0,C 180,E1 -29185.221,E2 -29185.221} C_VEL
LIN {X 0,Y 141.908,Z 911.565,A -85,B 0,C 180,E1 -29190.955,E2 -29190.955} C_VEL
LIN {X 0,Y 128.724,Z 921.492,A -85,B 0,C 180,E1 -29198.42,E2 -29198.42} C_VEL
LIN {X 0,Y 117.954,Z 929.505,A -85,B 0,C 180,E1 -29207.519,E2 -29207.519} C_VEL
LIN {X 0,Y 110.325,Z 935.758,A -85,B 0,C 180,E1 -29218.288,E2 -29218.288} C_VEL
LIN {X 0,Y 106.56,Z 940.214,A -85,B 0,C 180,E1 -29230.257,E2 -29230.257} C_VEL
LIN {X 0,Y 106.497,Z 942.645,A -85,B 0,C 180,E1 -29241.361,E2 -29241.361} C_VEL
LIN {X 0,Y 107.684,Z 943.393,A -85,B 0,C 180,E1 -29248.936,E2 -29248.936} C_VEL
LIN {X 0,Y 107.523,Z 943.304,A -85,B 0,C 180,E1 -29252.665,E2 -29252.665} C_VEL
LIN {X 0,Y 106.555,Z 942.128,A -85,B 0,C 180,E1 -29261.914,E2 -29261.914} C_VEL
LIN {X 0,Y 108.075,Z 939.083,A -85,B 0,C 180,E1 -29273.443,E2 -29273.443} C_VEL
LIN {X 0,Y 113.688,Z 934.082,A -85,B 0,C 180,E1 -29284.868,E2 -29284.868} C_VEL
LIN {X 0,Y 122.097,Z 928.266,A -85,B 0,C 180,E1 -29293.789,E2 -29293.789} C_VEL
LIN {X 0,Y 134.399,Z 927.526,A -85,B 0,C 180,E1 -29303.119,E2 -29303.119} C_VEL
LIN {X 0,Y 122.146,Z 919.286,A -85,B 0,C 180,E1 -29311.654,E2 -29311.654} C_VEL
LIN {X 0,Y 117.025,Z 914.146,A -85,B 0,C 180,E1 -29316.856,E2 -29316.856} C_VEL
LIN {X 0,Y 113.073,Z 912.173,A -85,B 0,C 180,E1 -29323.033,E2 -29323.033} C_VEL
LIN {X 0,Y 109.453,Z 907.385,A -85,B 0,C 180,E1 -29339.477,E2 -29339.477} C_VEL
LIN {X 0,Y 112.67,Z 903.773,A -85,B 0,C 180,E1 -29352.298,E2 -29352.298} C_VEL
LIN {X 0,Y 132.126,Z 896.959,A -85,B 0,C 180,E1 -29372.501,E2 -29372.501} C_VEL
LIN {X 0,Y 147.028,Z 893.272,A -85,B 0,C 180,E1 -29379.934,E2 -29379.934} C_VEL
LIN {X 0,Y 134.467,Z 901.254,A -85,B 0,C 180,E1 -29386.834,E2 -29386.834} C_VEL
LIN {X 0,Y 123.374,Z 907.709,A -85,B 0,C 180,E1 -29395.436,E2 -29395.436} C_VEL
LIN {X 0,Y 115.071,Z 912.271,A -85,B 0,C 180,E1 -29405.349,E2 -29405.349} C_VEL
LIN {X 0,Y 109.933,Z 915.057,A -85,B 0,C 180,E1 -29416.321,E2 -29416.321} C_VEL
LIN {X 0,Y 107.974,Z 916.152,A -85,B 0,C 180,E1 -29427.346,E2 -29427.346} C_VEL
LIN {X 0,Y 108.551,Z 915.84,A -85,B 0,C 180,E1 -29437.942,E2 -29437.942} C_VEL
LIN {X 0,Y 111.827,Z 914.064,A -85,B 0,C 180,E1 -29448.777,E2 -29448.777} C_VEL
LIN {X 0,Y 118.054,Z 910.725,A -85,B 0,C 180,E1 -29458.867,E2 -29458.867} C_VEL
LIN {X 0,Y 127.045,Z 905.724,A -85,B 0,C 180,E1 -29467.871,E2 -29467.871} C_VEL
LIN {X 0,Y 137.834,Z 899.315,A -85,B 0,C 180,E1 -29475.31,E2 -29475.31} C_VEL
LIN {X 0,Y 150.392,Z 891.155,A -85,B 0,C 180,E1 -29481.677,E2 -29481.677} C_VEL
LIN {X 0,Y 163.633,Z 881.615,A -85,B 0,C 180,E1 -29486.84,E2 -29486.84} C_VEL
LIN {X 0,Y 177.108,Z 870.743,A -85,B 0,C 180,E1 -29491.053,E2 -29491.053} C_VEL
LIN {X 0,Y 190.507,Z 858.582,A -85,B 0,C 180,E1 -29494.522,E2 -29494.522} C_VEL
LIN {X 0,Y 203.6,Z 845.135,A -85,B 0,C 180,E1 -29497.41,E2 -29497.41} C_VEL
LIN {X 0,Y 216.219,Z 830.357,A -85,B 0,C 180,E1 -29499.844,E2 -29499.844} C_VEL
LIN {X 0,Y 228.251,Z 814.145,A -85,B 0,C 180,E1 -29501.916,E2 -29501.916} C_VEL
LIN {X 0,Y 238.722,Z 797.816,A -85,B 0,C 180,E1 -29503.57,E2 -29503.57} C_VEL
LIN {X 0,Y 248.421,Z 780.045,A -85,B 0,C 180,E1 -29505.015,E2 -29505.015} C_VEL
LIN {X 0,Y 256.415,Z 762.648,A -85,B 0,C 180,E1 -29506.161,E2 -29506.161} C_VEL
LIN {X 0,Y 263.544,Z 743.638,A -85,B 0,C 180,E1 -29507.177,E2 -29507.177} C_VEL
LIN {X 0,Y 273.408,Z 710.345,A -85,B 0,C 180,E1 -29508.554,E2 -29508.554} C_VEL
LIN {X 0,Y 282.511,Z 675.791,A -85,B 0,C 180,E1 -29509.641,E2 -29509.641} C_VEL
